C09132=1213.052,331.512,-71.588,-176.205,7.411,148.299
C09133=1213.056,331.264,-71.557,-176.207,7.408,148.299
C09134=1213.060,331.016,-71.525,-176.210,7.405,148.299
C09135=1213.064,330.768,-71.494,-176.212,7.402,148.299
C09136=1213.068,330.520,-71.463,-176.214,7.400,148.299
C09137=1213.073,330.272,-71.431,-176.216,7.396,148.298
C09138=1213.077,330.024,-71.400,-176.218,7.394,148.299
C09139=1213.081,329.776,-71.369,-176.220,7.391,148.298
C09140=1213.085,329.528,-71.338,-176.223,7.389,148.298
C09141=1213.089,329.280,-71.306,-176.225,7.385,148.298
C09142=1213.093,329.032,-71.275,-176.227,7.383,148.298
C09143=1213.098,328.784,-71.243,-176.229,7.380,148.298
C09144=1213.102,328.536,-71.212,-176.231,7.378,148.298
C09145=1213.106,328.288,-71.182,-176.233,7.374,148.298
C09146=1213.111,328.040,-71.150,-176.235,7.372,148.298
C09147=1213.115,327.792,-71.119,-176.238,7.369,148.298
C09148=1213.119,327.544,-71.087,-176.240,7.366,148.298
C09149=1213.123,327.296,-71.056,-176.242,7.363,148.297
C09150=1213.128,327.048,-71.026,-176.245,7.360,148.297
C09151=1213.132,326.800,-70.994,-176.246,7.358,148.297
C09152=1213.136,326.552,-70.963,-176.249,7.354,148.297
C09153=1213.141,326.304,-70.932,-176.251,7.352,148.297
C09154=1213.144,326.056,-70.900,-176.253,7.349,148.297
C09155=1213.148,325.808,-70.870,-176.255,7.347,148.297
C09156=1213.153,325.560,-70.839,-176.258,7.343,148.297
C09157=1213.157,325.311,-70.808,-176.260,7.341,148.297
C09158=1213.161,325.064,-70.777,-176.262,7.338,148.297
C09159=1213.165,324.815,-70.746,-176.264,7.336,148.297
C09160=1213.170,324.568,-70.715,-176.267,7.333,148.297
C09161=1213.174,324.320,-70.684,-176.268,7.330,148.297
C09162=1213.178,324.071,-70.653,-176.271,7.327,148.297
C09163=1213.182,323.824,-70.622,-176.273,7.325,148.297
C09164=1213.186,323.576,-70.591,-176.275,7.321,148.296
C09165=1213.191,323.327,-70.560,-176.277,7.319,148.296
C09166=1213.195,323.079,-70.530,-176.280,7.316,148.296
C09167=1213.199,322.831,-70.498,-176.282,7.313,148.296
C09168=1213.203,322.583,-70.468,-176.284,7.311,148.296
C09169=1213.207,322.336,-70.437,-176.287,7.307,148.296
C09170=1213.211,322.087,-70.406,-176.289,7.305,148.296
C09171=1213.216,321.839,-70.375,-176.291,7.302,148.296
C09172=1213.221,321.591,-70.344,-176.293,7.299,148.296
C09173=1213.224,321.343,-70.314,-176.296,7.296,148.296
C09174=1213.228,321.095,-70.283,-176.298,7.294,148.296
C09175=1213.233,320.847,-70.252,-176.300,7.291,148.296
C09176=1213.238,320.599,-70.221,-176.302,7.289,148.296
C09177=1213.241,320.351,-70.191,-176.305,7.286,148.296
C09178=1213.246,320.103,-70.160,-176.307,7.283,148.296
C09179=1213.250,319.855,-70.129,-176.309,7.280,148.296
C09180=1213.254,319.606,-70.098,-176.311,7.278,148.296
C09181=1213.258,319.358,-70.068,-176.314,7.275,148.296
C09182=1213.263,319.110,-70.037,-176.316,7.272,148.296
C09183=1213.267,318.862,-70.006,-176.318,7.269,148.296
C09184=1213.271,318.614,-69.976,-176.320,7.267,148.296
C09185=1213.275,318.366,-69.945,-176.323,7.264,148.296
C09186=1213.280,318.118,-69.914,-176.325,7.262,148.295
C09187=1213.284,317.870,-69.884,-176.327,7.258,148.295
C09188=1213.288,317.622,-69.853,-176.330,7.255,148.295
C09189=1213.293,317.373,-69.823,-176.332,7.253,148.295
C09190=1213.296,317.126,-69.793,-176.334,7.250,148.295
C09191=1213.301,316.878,-69.762,-176.336,7.248,148.295
C09192=1213.305,316.629,-69.731,-176.339,7.245,148.295
C09193=1213.309,316.381,-69.701,-176.341,7.242,148.295
C09194=1213.314,316.133,-69.670,-176.343,7.239,148.295
C09195=1213.318,315.885,-69.641,-176.346,7.237,148.295
C09196=1213.322,315.637,-69.610,-176.348,7.234,148.295
C09197=1213.327,315.361,-69.575,-176.351,7.231,148.295
C09198=1213.332,315.084,-69.542,-176.354,7.228,148.295
C09199=1213.336,314.809,-69.508,-176.356,7.226,148.295
C09200=1213.341,314.532,-69.474,-176.358,7.222,148.295
C09201=1213.345,314.284,-69.444,-176.361,7.219,148.295
C09202=1213.349,314.037,-69.413,-176.363,7.217,148.295
C09203=1213.354,313.789,-69.383,-176.365,7.214,148.295
C09204=1213.358,313.541,-69.353,-176.368,7.212,148.295
C09205=1213.363,313.293,-69.322,-176.370,7.209,148.295
C09206=1213.366,313.044,-69.292,-176.372,7.206,148.295
C09207=1213.371,312.796,-69.262,-176.375,7.203,148.295
C09208=1213.375,312.548,-69.232,-176.377,7.201,148.295
C09209=1213.379,312.300,-69.201,-176.379,7.198,148.295
C09210=1213.384,312.052,-69.171,-176.381,7.196,148.295
C09211=1213.388,311.804,-69.141,-176.384,7.193,148.295
C09212=1213.392,311.556,-69.111,-176.386,7.190,148.295
C09213=1213.396,311.307,-69.080,-176.389,7.187,148.295
C09214=1213.400,311.059,-69.050,-176.392,7.184,148.295
C09215=1213.405,310.811,-69.020,-176.393,7.182,148.295
C09216=1213.409,310.563,-68.990,-176.396,7.179,148.295
C09217=1213.413,310.315,-68.960,-176.398,7.177,148.295
C09218=1213.418,310.067,-68.929,-176.401,7.173,148.295
C09219=1213.422,309.819,-68.900,-176.403,7.171,148.295
C09220=1213.427,309.571,-68.869,-176.405,7.168,148.295
C09221=1213.431,309.322,-68.840,-176.408,7.166,148.295
C09222=1213.435,309.074,-68.809,-176.410,7.163,148.295
C09223=1213.440,308.826,-68.780,-176.412,7.161,148.295
C09224=1213.443,308.578,-68.749,-176.415,7.158,148.295
C09225=1213.448,308.329,-68.719,-176.417,7.156,148.295
C09226=1213.452,308.081,-68.689,-176.419,7.152,148.295
C09227=1213.456,307.833,-68.659,-176.421,7.150,148.295
C09228=1213.461,307.585,-68.629,-176.424,7.147,148.295
C09229=1213.465,307.337,-68.599,-176.426,7.145,148.295
C09230=1213.469,307.089,-68.570,-176.429,7.142,148.295
C09231=1213.473,306.841,-68.539,-176.431,7.140,148.295
C09232=1213.478,306.593,-68.509,-176.433,7.137,148.295
C09233=1213.482,306.344,-68.480,-176.436,7.134,148.295
C09234=1213.486,306.096,-68.449,-176.438,7.132,148.295
C09235=1213.491,305.848,-68.420,-176.441,7.129,148.295
C09236=1213.495,305.600,-68.390,-176.443,7.127,148.295
C09237=1213.499,305.352,-68.360,-176.445,7.124,148.295
C09238=1213.504,305.104,-68.330,-176.448,7.122,148.296
C09239=1213.508,304.855,-68.301,-176.450,7.119,148.296
C09240=1213.512,304.607,-68.271,-176.452,7.116,148.296
C09241=1213.517,304.359,-68.240,-176.455,7.113,148.296
C09242=1213.521,304.111,-68.211,-176.457,7.111,148.296
C09243=1213.525,303.862,-68.182,-176.460,7.108,148.296
C09244=1213.529,303.614,-68.152,-176.462,7.106,148.296
C09245=1213.534,303.366,-68.121,-176.465,7.103,148.296
C09246=1213.538,303.118,-68.092,-176.467,7.101,148.296
C09247=1213.542,302.870,-68.062,-176.469,7.098,148.296
C09248=1213.546,302.621,-68.033,-176.472,7.095,148.296
C09249=1213.550,302.373,-68.004,-176.474,7.092,148.296
C09250=1213.555,302.125,-67.973,-176.476,7.090,148.296
C09251=1213.559,301.877,-67.943,-176.479,7.087,148.296
C09252=1213.563,301.629,-67.914,-176.481,7.085,148.296
C09253=1213.568,301.380,-67.884,-176.484,7.082,148.296
C09254=1213.572,301.132,-67.855,-176.486,7.080,148.296
C09255=1213.577,300.885,-67.826,-176.489,7.077,148.296
C09256=1213.581,300.636,-67.796,-176.491,7.074,148.296
C09257=1213.586,300.388,-67.766,-176.494,7.072,148.296
C09258=1213.590,300.139,-67.737,-176.496,7.069,148.296
C09259=1213.594,299.891,-67.707,-176.498,7.067,148.297
C09260=1213.598,299.643,-67.678,-176.501,7.064,148.297
C09261=1213.602,299.395,-67.649,-176.503,7.062,148.297
C09262=1213.607,299.146,-67.619,-176.506,7.059,148.297
C09263=1213.611,298.898,-67.590,-176.508,7.057,148.297
C09264=1213.615,298.650,-67.560,-176.510,7.054,148.297
C09265=1213.619,298.402,-67.531,-176.513,7.052,148.297
C09266=1213.624,298.154,-67.502,-176.515,7.049,148.297
C09267=1213.628,297.906,-67.472,-176.517,7.046,148.297
C09268=1213.632,297.658,-67.443,-176.520,7.043,148.297
C09269=1213.636,297.409,-67.413,-176.523,7.041,148.297
C09270=1213.641,297.161,-67.383,-176.525,7.038,148.297
C09271=1213.646,296.912,-67.354,-176.527,7.036,148.297
C09272=1213.650,296.664,-67.324,-176.530,7.034,148.297
C09273=1213.655,296.416,-67.296,-176.532,7.031,148.297
C09274=1213.659,296.168,-67.267,-176.534,7.029,148.297
C09275=1213.662,295.920,-67.238,-176.537,7.026,148.297
C09276=1213.667,295.671,-67.208,-176.539,7.023,148.297
C09277=1213.671,295.423,-67.179,-176.542,7.021,148.298
C09278=1213.675,295.175,-67.149,-176.544,7.019,148.298
C09279=1213.679,294.926,-67.121,-176.547,7.016,148.298
C09280=1213.684,294.678,-67.091,-176.549,7.013,148.298
C09281=1213.688,294.430,-67.062,-176.551,7.011,148.298
C09282=1213.693,294.182,-67.033,-176.554,7.008,148.298
C09283=1213.697,293.934,-67.003,-176.557,7.006,148.298
C09284=1213.701,293.685,-66.974,-176.559,7.003,148.298
C09285=1213.706,293.437,-66.945,-176.561,7.001,148.298
C09286=1213.710,293.189,-66.916,-176.564,6.998,148.298
C09287=1213.715,292.940,-66.887,-176.566,6.996,148.298
C09288=1213.719,292.692,-66.858,-176.568,6.994,148.298
C09289=1213.723,292.445,-66.829,-176.572,6.991,148.299
C09290=1213.727,292.196,-66.800,-176.574,6.989,148.299
C09291=1213.732,291.947,-66.771,-176.576,6.986,148.299
C09292=1213.736,291.699,-66.741,-176.578,6.983,148.299
C09293=1213.740,291.450,-66.713,-176.581,6.980,148.299
C09294=1213.745,291.203,-66.684,-176.583,6.978,148.299
C09295=1213.748,290.955,-66.655,-176.586,6.976,148.299
C09296=1213.753,290.706,-66.626,-176.589,6.973,148.299
C09297=1213.757,290.458,-66.597,-176.591,6.971,148.299
C09298=1213.762,290.209,-66.568,-176.593,6.968,148.299
C09299=1213.766,289.961,-66.539,-176.596,6.966,148.300
C09300=1213.771,289.713,-66.509,-176.599,6.963,148.300
C09301=1213.775,289.438,-66.478,-176.601,6.961,148.300
C09302=1213.780,289.164,-66.446,-176.603,6.958,148.300
C09303=1213.785,288.890,-66.414,-176.607,6.955,148.300
C09304=1213.790,288.616,-66.382,-176.609,6.952,148.300
C09305=1213.795,288.368,-66.354,-176.611,6.950,148.300
C09306=1213.798,288.120,-66.325,-176.614,6.948,148.300
C09307=1213.803,287.871,-66.296,-176.617,6.945,148.300
C09308=1213.808,287.623,-66.268,-176.619,6.943,148.300
C09309=1213.812,287.375,-66.238,-176.621,6.940,148.300
C09310=1213.816,287.126,-66.210,-176.624,6.938,148.301
C09311=1213.820,286.878,-66.181,-176.626,6.936,148.301
C09312=1213.825,286.629,-66.152,-176.629,6.933,148.301
C09313=1213.828,286.382,-66.123,-176.631,6.930,148.301
C09314=1213.833,286.133,-66.095,-176.634,6.928,148.301
C09315=1213.838,285.884,-66.066,-176.636,6.925,148.301
C09316=1213.841,285.637,-66.037,-176.638,6.923,148.301
C09317=1213.846,285.388,-66.009,-176.642,6.921,148.301
C09318=1213.851,285.139,-65.980,-176.644,6.918,148.301
C09319=1213.854,284.891,-65.952,-176.646,6.915,148.301
C09320=1213.859,284.643,-65.923,-176.648,6.913,148.302
C09321=1213.864,284.394,-65.894,-176.651,6.911,148.302
C09322=1213.867,284.146,-65.866,-176.654,6.908,148.302
C09323=1213.872,283.898,-65.837,-176.656,6.906,148.302
C09324=1213.876,283.650,-65.809,-176.659,6.903,148.302
C09325=1213.881,283.402,-65.781,-176.661,6.901,148.302
C09326=1213.885,283.153,-65.751,-176.663,6.899,148.302
C09327=1213.889,282.905,-65.723,-176.666,6.896,148.302
C09328=1213.894,282.656,-65.695,-176.669,6.894,148.303
C09329=1213.898,282.408,-65.667,-176.671,6.892,148.303
C09330=1213.903,282.160,-65.638,-176.673,6.889,148.303
C09331=1213.907,281.912,-65.609,-176.676,6.887,148.303
C09332=1213.912,281.664,-65.581,-176.679,6.884,148.303
C09333=1213.916,281.415,-65.552,-176.681,6.882,148.303
C09334=1213.920,281.166,-65.524,-176.683,6.880,148.303
C09335=1213.925,280.918,-65.496,-176.686,6.877,148.303
C09336=1213.929,280.669,-65.468,-176.688,6.875,148.304
C09337=1213.934,280.421,-65.439,-176.691,6.873,148.304
C09338=1213.938,280.173,-65.411,-176.694,6.870,148.304
C09339=1213.942,279.925,-65.382,-176.696,6.867,148.304
C09340=1213.946,279.676,-65.354,-176.698,6.866,148.304
C09341=1213.950,279.429,-65.326,-176.701,6.863,148.304
C09342=1213.955,279.180,-65.297,-176.703,6.860,148.304
C09343=1213.959,278.932,-65.270,-176.706,6.858,148.305
C09344=1213.964,278.683,-65.241,-176.708,6.855,148.305
C09345=1213.968,278.435,-65.213,-176.710,6.853,148.305
C09346=1213.973,278.186,-65.184,-176.714,6.851,148.305
C09347=1213.977,277.938,-65.156,-176.716,6.848,148.305
C09348=1213.981,277.689,-65.128,-176.718,6.846,148.305
C09349=1213.986,277.442,-65.100,-176.721,6.843,148.305
C09350=1213.990,277.193,-65.072,-176.723,6.841,148.305
C09351=1213.995,276.945,-65.043,-176.726,6.839,148.306
C09352=1213.998,276.696,-65.015,-176.728,6.836,148.306
C09353=1214.003,276.448,-64.988,-176.731,6.834,148.306
C09354=1214.008,276.199,-64.960,-176.733,6.832,148.306
C09355=1214.012,275.951,-64.932,-176.736,6.829,148.306
C09356=1214.016,275.702,-64.903,-176.739,6.827,148.306
C09357=1214.021,275.454,-64.875,-176.741,6.825,148.306
C09358=1214.024,275.206,-64.847,-176.743,6.822,148.307
C09359=1214.030,274.957,-64.819,-176.746,6.820,148.307
C09360=1214.033,274.709,-64.791,-176.748,6.818,148.307
C09361=1214.038,274.460,-64.763,-176.751,6.815,148.307
C09362=1214.043,274.212,-64.735,-176.753,6.813,148.307
C09363=1214.047,273.964,-64.707,-176.755,6.811,148.307
C09364=1214.051,273.716,-64.679,-176.759,6.808,148.308
C09365=1214.055,273.467,-64.651,-176.761,6.806,148.308
C09366=1214.060,273.218,-64.623,-176.763,6.804,148.308
C09367=1214.064,272.970,-64.595,-176.766,6.801,148.308
C09368=1214.068,272.722,-64.567,-176.768,6.799,148.308
C09369=1214.073,272.474,-64.539,-176.771,6.797,148.308
C09370=1214.078,272.224,-64.512,-176.773,6.794,148.308
C09371=1214.082,271.977,-64.484,-176.776,6.792,148.309
C09372=1214.086,271.728,-64.456,-176.778,6.790,148.309
C09373=1214.090,271.480,-64.429,-176.781,6.788,148.309
C09374=1214.095,271.231,-64.400,-176.784,6.785,148.309
C09375=1214.099,270.983,-64.372,-176.786,6.783,148.309
C09376=1214.104,270.734,-64.345,-176.788,6.781,148.309
C09377=1214.108,270.486,-64.317,-176.791,6.778,148.309
C09378=1214.112,270.238,-64.289,-176.794,6.776,148.310
C09379=1214.117,269.989,-64.262,-176.796,6.774,148.310
C09380=1214.122,269.741,-64.234,-176.799,6.771,148.310
C09381=1214.126,269.492,-64.206,-176.801,6.769,148.310
C09382=1214.130,269.244,-64.179,-176.804,6.767,148.310
C09383=1214.134,268.996,-64.151,-176.806,6.765,148.311
C09384=1214.138,268.747,-64.123,-176.809,6.762,148.311
C09385=1214.144,268.499,-64.095,-176.811,6.760,148.311
C09386=1214.148,268.250,-64.068,-176.814,6.758,148.311
C09387=1214.152,268.002,-64.040,-176.816,6.755,148.311
C09388=1214.157,267.753,-64.013,-176.818,6.753,148.311
C09389=1214.161,267.505,-63.985,-176.821,6.751,148.312
C09390=1214.165,267.256,-63.958,-176.823,6.749,148.312
C09391=1214.169,267.008,-63.930,-176.826,6.746,148.312
C09392=1214.174,266.760,-63.903,-176.828,6.744,148.312
C09393=1214.178,266.511,-63.875,-176.831,6.742,148.312
C09394=1214.183,266.262,-63.847,-176.834,6.739,148.312
C09395=1214.188,266.015,-63.819,-176.836,6.737,148.313
C09396=1214.192,265.766,-63.792,-176.839,6.735,148.313
C09397=1214.196,265.517,-63.765,-176.841,6.733,148.313
C09398=1214.201,265.269,-63.737,-176.844,6.730,148.313
C09399=1214.205,265.020,-63.710,-176.846,6.728,148.313
C09400=1214.210,264.772,-63.683,-176.849,6.726,148.313
C09401=1214.214,264.523,-63.655,-176.851,6.724,148.314
C09402=1214.218,264.275,-63.628,-176.854,6.721,148.314
C09403=1214.223,264.027,-63.600,-176.856,6.719,148.314
C09404=1214.227,263.779,-63.573,-176.859,6.717,148.314
C09405=1214.231,263.505,-63.543,-176.862,6.714,148.314
C09406=1214.236,263.233,-63.512,-176.864,6.712,148.315
C09407=1214.241,262.960,-63.483,-176.867,6.709,148.315
C09408=1214.247,262.687,-63.453,-176.870,6.708,148.315
C09409=1214.251,262.439,-63.425,-176.873,6.705,148.315
C09410=1214.255,262.190,-63.398,-176.875,6.703,148.315
C09411=1214.260,261.942,-63.371,-176.878,6.701,148.316
C09412=1214.264,261.693,-63.344,-176.880,6.699,148.316
C09413=1214.269,261.445,-63.317,-176.883,6.696,148.316
C09414=1214.273,261.197,-63.289,-176.885,6.694,148.316
C09415=1214.277,260.948,-63.262,-176.888,6.692,148.316
C09416=1214.281,260.700,-63.235,-176.890,6.690,148.316
C09417=1214.286,260.451,-63.208,-176.893,6.687,148.317
C09418=1214.291,260.203,-63.181,-176.895,6.685,148.317
C09419=1214.295,259.955,-63.153,-176.898,6.683,148.317
C09420=1214.300,259.706,-63.126,-176.900,6.681,148.317
C09421=1214.304,259.457,-63.099,-176.903,6.678,148.317
C09422=1214.308,259.209,-63.072,-176.906,6.676,148.318
C09423=1214.312,258.960,-63.045,-176.908,6.674,148.318
C09424=1214.317,258.712,-63.018,-176.910,6.672,148.318
C09425=1214.322,258.463,-62.991,-176.913,6.670,148.318
C09426=1214.326,258.215,-62.964,-176.916,6.667,148.319
C09427=1214.331,257.966,-62.937,-176.918,6.665,148.319
C09428=1214.334,257.717,-62.910,-176.920,6.663,148.319
C09429=1214.339,257.469,-62.883,-176.923,6.661,148.319
C09430=1214.344,257.220,-62.856,-176.925,6.659,148.319
C09431=1214.348,256.972,-62.829,-176.928,6.656,148.320
C09432=1214.353,256.723,-62.802,-176.931,6.654,148.320
C09433=1214.357,256.475,-62.775,-176.933,6.652,148.320
C09434=1214.361,256.227,-62.748,-176.935,6.650,148.320
C09435=1214.366,255.978,-62.721,-176.938,6.647,148.320
C09436=1214.371,255.730,-62.694,-176.941,6.646,148.321
C09437=1214.375,255.482,-62.668,-176.943,6.643,148.321
C09438=1214.379,255.232,-62.640,-176.946,6.641,148.321
C09439=1214.383,254.984,-62.613,-176.948,6.639,148.321
C09440=1214.387,254.736,-62.587,-176.951,6.637,148.321
C09441=1214.392,254.487,-62.560,-176.954,6.635,148.322
C09442=1214.397,254.239,-62.532,-176.956,6.633,148.322
C09443=1214.401,253.990,-62.505,-176.958,6.631,148.322
C09444=1214.405,253.741,-62.480,-176.961,6.628,148.322
C09445=1214.410,253.493,-62.453,-176.963,6.627,148.322
C09446=1214.415,253.244,-62.426,-176.966,6.624,148.323
C09447=1214.419,252.996,-62.399,-176.969,6.622,148.323
C09448=1214.423,252.748,-62.372,-176.971,6.620,148.323
C09449=1214.428,252.499,-62.345,-176.973,6.618,148.323
C09450=1214.432,252.250,-62.319,-176.976,6.616,148.324
C09451=1214.437,252.002,-62.292,-176.979,6.613,148.324
C09452=1214.441,251.754,-62.266,-176.981,6.611,148.324
C09453=1214.445,251.505,-62.239,-176.984,6.609,148.324
C09454=1214.450,251.256,-62.212,-176.986,6.607,148.324
C09455=1214.454,251.008,-62.186,-176.989,6.605,148.325
C09456=1214.459,250.759,-62.159,-176.991,6.603,148.325
C09457=1214.463,250.511,-62.132,-176.994,6.600,148.325
C09458=1214.468,250.262,-62.106,-176.997,6.598,148.325
C09459=1214.473,250.014,-62.079,-176.999,6.596,148.326
C09460=1214.476,249.765,-62.052,-177.001,6.594,148.326
C09461=1214.481,249.516,-62.026,-177.004,6.592,148.326
C09462=1214.485,249.268,-62.000,-177.007,6.590,148.326
C09463=1214.490,249.020,-61.973,-177.009,6.587,148.326
C09464=1214.494,248.771,-61.947,-177.012,6.586,148.327
C09465=1214.499,248.522,-61.920,-177.014,6.584,148.327
C09466=1214.503,248.274,-61.894,-177.017,6.582,148.327
C09467=1214.508,248.025,-61.867,-177.019,6.580,148.327
C09468=1214.512,247.777,-61.840,-177.022,6.578,148.328
C09469=1214.517,247.528,-61.814,-177.024,6.576,148.328
C09470=1214.521,247.280,-61.788,-177.027,6.573,148.328
C09471=1214.526,247.030,-61.761,-177.030,6.571,148.328
C09472=1214.529,246.782,-61.735,-177.032,6.569,148.328
C09473=1214.535,246.534,-61.709,-177.035,6.567,148.329
C09474=1214.539,246.286,-61.682,-177.037,6.565,148.329
C09475=1214.544,246.037,-61.656,-177.039,6.563,148.329
C09476=1214.548,245.788,-61.630,-177.042,6.561,148.329
C09477=1214.553,245.539,-61.603,-177.045,6.558,148.330
C09478=1214.557,245.291,-61.577,-177.047,6.556,148.330
C09479=1214.561,245.042,-61.551,-177.050,6.554,148.330
C09480=1214.566,244.794,-61.524,-177.053,6.552,148.330
C09481=1214.570,244.545,-61.498,-177.055,6.550,148.331
C09482=1214.574,244.296,-61.471,-177.057,6.548,148.331
C09483=1214.579,244.048,-61.446,-177.060,6.547,148.331
C09484=1214.583,243.800,-61.420,-177.063,6.544,148.331
C09485=1214.588,243.551,-61.393,-177.065,6.542,148.332
C09486=1214.592,243.302,-61.367,-177.068,6.540,148.332
C09487=1214.597,243.054,-61.340,-177.070,6.538,148.332
C09488=1214.601,242.805,-61.314,-177.073,6.536,148.332
C09489=1214.605,242.556,-61.289,-177.075,6.534,148.333
C09490=1214.611,242.308,-61.262,-177.078,6.532,148.333
C09491=1214.615,242.060,-61.236,-177.080,6.530,148.333
C09492=1214.619,241.811,-61.210,-177.083,6.528,148.333
C09493=1214.624,241.562,-61.183,-177.086,6.525,148.334
C09494=1214.628,241.313,-61.158,-177.088,6.523,148.334
C09495=1214.632,241.065,-61.132,-177.091,6.521,148.334
C09496=1214.637,240.817,-61.106,-177.093,6.519,148.334
C09497=1214.642,240.568,-61.079,-177.096,6.518,148.335
C09498=1214.646,240.319,-61.054,-177.098,6.515,148.335
C09499=1214.650,240.070,-61.028,-177.101,6.514,148.335
C09500=1214.655,239.821,-61.002,-177.103,6.512,148.335
C09501=1214.660,239.574,-60.975,-177.105,6.509,148.335
C09502=1214.664,239.325,-60.950,-177.109,6.507,148.336
C09503=1214.668,239.076,-60.924,-177.111,6.505,148.336
C09504=1214.673,238.827,-60.898,-177.114,6.503,148.336
C09505=1214.677,238.578,-60.872,-177.116,6.501,148.336
C09506=1214.682,238.330,-60.846,-177.119,6.499,148.337
C09507=1214.686,238.082,-60.820,-177.121,6.497,148.337
C09508=1214.690,237.833,-60.794,-177.124,6.495,148.337
C09509=1214.696,237.562,-60.766,-177.126,6.493,148.337
C09510=1214.701,237.290,-60.738,-177.129,6.490,148.338
C09511=1214.705,237.019,-60.709,-177.132,6.489,148.338
C09512=1214.711,236.747,-60.682,-177.135,6.486,148.338
C09513=1214.715,236.499,-60.656,-177.138,6.484,148.339
C09514=1214.719,236.250,-60.630,-177.140,6.482,148.339
C09515=1214.724,236.002,-60.605,-177.142,6.480,148.339
C09516=1214.728,235.753,-60.579,-177.145,6.478,148.339
C09517=1214.733,235.504,-60.553,-177.148,6.476,148.340
C09518=1214.737,235.255,-60.527,-177.150,6.474,148.340
C09519=1214.742,235.007,-60.501,-177.152,6.472,148.340
C09520=1214.746,234.758,-60.476,-177.155,6.470,148.340
C09521=1214.751,234.509,-60.450,-177.158,6.469,148.341
C09522=1214.755,234.261,-60.425,-177.160,6.467,148.341
C09523=1214.760,234.012,-60.399,-177.163,6.465,148.341
C09524=1214.764,233.763,-60.373,-177.165,6.463,148.342
C09525=1214.769,233.515,-60.348,-177.168,6.460,148.342
C09526=1214.773,233.267,-60.322,-177.171,6.458,148.342
C09527=1214.778,233.017,-60.296,-177.173,6.456,148.342
C09528=1214.783,232.769,-60.270,-177.176,6.454,148.343
C09529=1214.787,232.521,-60.244,-177.178,6.452,148.343
C09530=1214.791,232.272,-60.219,-177.181,6.450,148.343
C09531=1214.796,232.024,-60.193,-177.183,6.448,148.344
C09532=1214.800,231.775,-60.167,-177.186,6.447,148.344
C09533=1214.805,231.525,-60.142,-177.188,6.444,148.344
C09534=1214.810,231.277,-60.117,-177.191,6.443,148.344
C09535=1214.814,231.029,-60.091,-177.193,6.441,148.345
C09536=1214.818,230.780,-60.066,-177.196,6.439,148.345
C09537=1214.823,230.532,-60.040,-177.199,6.437,148.345
C09538=1214.827,230.282,-60.015,-177.201,6.435,148.345
C09539=1214.832,230.033,-59.989,-177.204,6.433,148.346
C09540=1214.837,229.785,-59.964,-177.206,6.431,148.346
C09541=1214.841,229.536,-59.938,-177.209,6.429,148.346
C09542=1214.846,229.288,-59.913,-177.211,6.427,148.347
C09543=1214.850,229.039,-59.888,-177.214,6.425,148.347
C09544=1214.854,228.790,-59.863,-177.216,6.423,148.347
C09545=1214.858,228.542,-59.837,-177.219,6.421,148.347
C09546=1214.863,228.293,-59.812,-177.222,6.419,148.348
C09547=1214.868,228.045,-59.787,-177.225,6.417,148.348
C09548=1214.872,227.796,-59.761,-177.227,6.415,148.348
C09549=1214.877,227.547,-59.736,-177.229,6.413,148.348
C09550=1214.881,227.298,-59.711,-177.232,6.411,148.349
C09551=1214.886,227.050,-59.685,-177.235,6.409,148.349
C09552=1214.891,226.801,-59.660,-177.237,6.407,148.349
C09553=1214.895,226.552,-59.635,-177.240,6.406,148.350
C09554=1214.899,226.304,-59.610,-177.243,6.404,148.350
C09555=1214.904,226.055,-59.585,-177.245,6.402,148.350
C09556=1214.908,225.807,-59.559,-177.247,6.400,148.350
C09557=1214.913,225.557,-59.534,-177.250,6.398,148.351
C09558=1214.918,225.309,-59.509,-177.253,6.396,148.351
C09559=1214.922,225.060,-59.483,-177.255,6.394,148.351
C09560=1214.926,224.812,-59.459,-177.258,6.392,148.352
C09561=1214.931,224.563,-59.433,-177.260,6.390,148.352
C09562=1214.936,224.315,-59.409,-177.263,6.388,148.352
C09563=1214.940,224.066,-59.383,-177.265,6.386,148.353
C09564=1214.945,223.817,-59.358,-177.268,6.385,148.353
C09565=1214.949,223.569,-59.333,-177.271,6.383,148.353
C09566=1214.954,223.320,-59.308,-177.273,6.381,148.354
C09567=1214.958,223.071,-59.283,-177.276,6.379,148.354
C09568=1214.963,222.822,-59.258,-177.278,6.377,148.354
C09569=1214.967,222.573,-59.232,-177.281,6.375,148.354
C09570=1214.972,222.325,-59.208,-177.283,6.373,148.355
C09571=1214.976,222.076,-59.183,-177.286,6.371,148.355
C09572=1214.981,221.828,-59.158,-177.288,6.369,148.355
C09573=1214.985,221.578,-59.133,-177.291,6.368,148.356
C09574=1214.990,221.330,-59.108,-177.294,6.366,148.356
C09575=1214.994,221.081,-59.083,-177.296,6.364,148.356
C09576=1214.999,220.832,-59.058,-177.299,6.362,148.356
C09577=1215.003,220.584,-59.033,-177.301,6.360,148.357
C09578=1215.008,220.335,-59.008,-177.304,6.358,148.357
C09579=1215.012,220.086,-58.983,-177.306,6.356,148.357
C09580=1215.017,219.838,-58.959,-177.309,6.354,148.358
C09581=1215.022,219.589,-58.934,-177.312,6.352,148.358
C09582=1215.026,219.340,-58.909,-177.314,6.351,148.358
C09583=1215.030,219.092,-58.884,-177.317,6.349,148.359
C09584=1215.035,218.842,-58.859,-177.320,6.347,148.359
C09585=1215.039,218.594,-58.835,-177.322,6.345,148.359
C09586=1215.044,218.346,-58.810,-177.324,6.343,148.359
C09587=1215.049,218.096,-58.785,-177.327,6.341,148.360
C09588=1215.053,217.848,-58.760,-177.330,6.339,148.360
C09589=1215.057,217.599,-58.735,-177.332,6.337,148.360
C09590=1215.062,217.350,-58.710,-177.335,6.336,148.361
C09591=1215.067,217.102,-58.686,-177.338,6.334,148.361
C09592=1215.071,216.853,-58.661,-177.340,6.332,148.361
C09593=1215.076,216.604,-58.637,-177.343,6.330,148.362
C09594=1215.080,216.355,-58.612,-177.345,6.328,148.362
C09595=1215.085,216.106,-58.588,-177.348,6.326,148.362
C09596=1215.089,215.858,-58.562,-177.350,6.324,148.363
C09597=1215.093,215.609,-58.538,-177.353,6.322,148.363
C09598=1215.098,215.360,-58.513,-177.356,6.320,148.363
C09599=1215.103,215.112,-58.489,-177.358,6.319,148.364
C09600=1215.107,214.863,-58.464,-177.361,6.317,148.364
C09601=1215.112,214.614,-58.439,-177.363,6.315,148.364
C09602=1215.117,214.365,-58.415,-177.366,6.313,148.365
C09603=1215.121,214.116,-58.390,-177.369,6.311,148.365
C09604=1215.126,213.868,-58.366,-177.371,6.309,148.365
C09605=1215.130,213.620,-58.341,-177.374,6.308,148.366
C09606=1215.134,213.370,-58.316,-177.377,6.306,148.366
C09607=1215.139,213.122,-58.292,-177.379,6.304,148.366
C09608=1215.144,212.873,-58.268,-177.382,6.302,148.367
C09609=1215.148,212.624,-58.243,-177.385,6.300,148.367
C09610=1215.153,212.375,-58.219,-177.387,6.298,148.367
C09611=1215.157,212.127,-58.195,-177.390,6.296,148.368
C09612=1215.162,211.878,-58.170,-177.392,6.295,148.368
C09613=1215.167,211.607,-58.144,-177.395,6.293,148.368
C09614=1215.172,211.337,-58.117,-177.398,6.291,148.369
C09615=1215.177,211.067,-58.091,-177.400,6.289,148.369
C09616=1215.182,210.797,-58.064,-177.403,6.287,148.369
C09617=1215.186,210.548,-58.040,-177.406,6.285,148.370
C09618=1215.191,210.298,-58.016,-177.408,6.284,148.370
C09619=1215.195,210.050,-57.992,-177.411,6.282,148.370
C09620=1215.201,209.801,-57.967,-177.414,6.280,148.371
C09621=1215.204,209.552,-57.942,-177.416,6.278,148.371
C09622=1215.209,209.304,-57.918,-177.419,6.276,148.371
C09623=1215.214,209.055,-57.894,-177.422,6.274,148.372
C09624=1215.218,208.806,-57.870,-177.424,6.272,148.372
C09625=1215.223,208.558,-57.846,-177.427,6.271,148.372
C09626=1215.228,208.308,-57.821,-177.429,6.269,148.373
C09627=1215.232,208.060,-57.797,-177.432,6.267,148.373
C09628=1215.236,207.811,-57.773,-177.435,6.265,148.373
C09629=1215.241,207.562,-57.748,-177.437,6.263,148.374
C09630=1215.245,207.313,-57.724,-177.439,6.262,148.374
C09631=1215.250,207.064,-57.701,-177.442,6.260,148.374
C09632=1215.255,206.815,-57.676,-177.445,6.259,148.375
C09633=1215.259,206.567,-57.652,-177.447,6.257,148.375
C09634=1215.264,206.318,-57.628,-177.450,6.255,148.375
C09635=1215.269,206.070,-57.604,-177.452,6.253,148.375
C09636=1215.273,205.820,-57.579,-177.455,6.251,148.376
C09637=1215.277,205.572,-57.555,-177.457,6.249,148.376
C09638=1215.282,205.323,-57.532,-177.460,6.247,148.376
C09639=1215.287,205.074,-57.508,-177.463,6.245,148.377
C09640=1215.292,204.826,-57.483,-177.465,6.244,148.377
C09641=1215.296,204.577,-57.460,-177.468,6.242,148.377
C09642=1215.300,204.327,-57.435,-177.470,6.241,148.378
C09643=1215.305,204.079,-57.411,-177.473,6.239,148.378
C09644=1215.309,203.830,-57.388,-177.475,6.237,148.378
C09645=1215.314,203.581,-57.363,-177.478,6.235,148.379
C09646=1215.319,203.332,-57.340,-177.481,6.233,148.379
C09647=1215.324,203.084,-57.316,-177.483,6.232,148.379
C09648=1215.328,202.835,-57.292,-177.486,6.230,148.380
C09649=1215.332,202.586,-57.268,-177.489,6.228,148.380
C09650=1215.337,202.337,-57.243,-177.491,6.226,148.381
C09651=1215.342,202.088,-57.220,-177.494,6.224,148.381
C09652=1215.346,201.840,-57.196,-177.496,6.223,148.381
C09653=1215.351,201.591,-57.173,-177.499,6.222,148.382
C09654=1215.355,201.342,-57.149,-177.502,6.220,148.382
C09655=1215.360,201.093,-57.125,-177.504,6.218,148.382
C09656=1215.364,200.845,-57.101,-177.507,6.216,148.383
C09657=1215.369,200.596,-57.078,-177.510,6.214,148.383
C09658=1215.374,200.347,-57.053,-177.512,6.212,148.384
C09659=1215.378,200.097,-57.029,-177.515,6.211,148.384
C09660=1215.383,199.849,-57.005,-177.517,6.210,148.384
C09661=1215.387,199.600,-56.982,-177.520,6.208,148.385
C09662=1215.392,199.351,-56.958,-177.522,6.206,148.385
C09663=1215.397,199.102,-56.934,-177.525,6.204,148.385
C09664=1215.401,198.854,-56.910,-177.528,6.202,148.386
C09665=1215.406,198.605,-56.887,-177.530,6.200,148.386
C09666=1215.410,198.356,-56.864,-177.533,6.199,148.386
C09667=1215.415,198.107,-56.840,-177.536,6.197,148.387
C09668=1215.419,197.858,-56.816,-177.538,6.196,148.387
C09669=1215.424,197.609,-56.793,-177.540,6.194,148.387
C09670=1215.429,197.361,-56.769,-177.543,6.192,148.388
C09671=1215.433,197.112,-56.745,-177.546,6.190,148.388
C09672=1215.438,196.863,-56.722,-177.548,6.188,148.388
C09673=1215.442,196.614,-56.698,-177.551,6.187,148.389
C09674=1215.447,196.365,-56.675,-177.554,6.185,148.389
C09675=1215.452,196.116,-56.651,-177.556,6.184,148.389
C09676=1215.456,195.868,-56.627,-177.558,6.182,148.390
C09677=1215.461,195.619,-56.604,-177.561,6.180,148.390
C09678=1215.466,195.370,-56.580,-177.564,6.178,148.390
C09679=1215.470,195.121,-56.557,-177.567,6.177,148.391
C09680=1215.475,194.872,-56.533,-177.569,6.175,148.391
C09681=1215.479,194.623,-56.510,-177.572,6.173,148.392
C09682=1215.484,194.374,-56.486,-177.574,6.172,148.392
C09683=1215.489,194.125,-56.463,-177.577,6.170,148.392
C09684=1215.493,193.876,-56.440,-177.579,6.168,148.393
C09685=1215.498,193.628,-56.416,-177.582,6.167,148.393
C09686=1215.502,193.379,-56.393,-177.585,6.165,148.394
C09687=1215.506,193.130,-56.369,-177.587,6.163,148.394
C09688=1215.511,192.881,-56.346,-177.589,6.162,148.394
C09689=1215.516,192.632,-56.323,-177.592,6.160,148.395
C09690=1215.521,192.383,-56.299,-177.595,6.158,148.395
C09691=1215.525,192.135,-56.275,-177.597,6.156,148.395
C09692=1215.530,191.886,-56.252,-177.600,6.155,148.396
C09693=1215.535,191.637,-56.229,-177.603,6.154,148.396
C09694=1215.539,191.389,-56.206,-177.605,6.152,148.397
C09695=1215.544,191.140,-56.183,-177.608,6.150,148.397
C09696=1215.548,190.891,-56.159,-177.610,6.148,148.397
C09697=1215.553,190.641,-56.136,-177.613,6.147,148.398
C09698=1215.558,190.392,-56.113,-177.616,6.145,148.398
C09699=1215.562,190.143,-56.089,-177.618,6.144,148.398
C09700=1215.566,189.895,-56.067,-177.621,6.142,148.399
C09701=1215.571,189.646,-56.043,-177.623,6.140,148.399
C09702=1215.576,189.397,-56.020,-177.626,6.138,148.399
C09703=1215.581,189.148,-55.997,-177.628,6.136,148.400
C09704=1215.585,188.900,-55.974,-177.631,6.135,148.400
C09705=1215.590,188.651,-55.951,-177.634,6.134,148.401
C09706=1215.594,188.402,-55.927,-177.636,6.132,148.401
C09707=1215.599,188.152,-55.904,-177.639,6.130,148.401
C09708=1215.603,187.904,-55.881,-177.642,6.128,148.402
C09709=1215.608,187.655,-55.858,-177.644,6.127,148.402
C09710=1215.613,187.406,-55.835,-177.646,6.126,148.402
C09711=1215.618,187.157,-55.812,-177.649,6.124,148.403
C09712=1215.622,186.909,-55.789,-177.652,6.122,148.403
C09713=1215.626,186.660,-55.765,-177.654,6.120,148.404
C09714=1215.631,186.410,-55.743,-177.657,6.119,148.404
C09715=1215.635,186.161,-55.720,-177.660,6.118,148.404
C09716=1215.641,185.913,-55.697,-177.662,6.116,148.405
C09717=1215.646,185.643,-55.672,-177.665,6.114,148.405
C09718=1215.651,185.374,-55.648,-177.668,6.112,148.406
C09719=1215.656,185.104,-55.623,-177.671,6.111,148.406
C09720=1215.661,184.835,-55.597,-177.673,6.109,148.406
C09721=1215.665,184.585,-55.575,-177.676,6.107,148.407
C09722=1215.670,184.336,-55.551,-177.679,6.105,148.407
C09723=1215.675,184.087,-55.528,-177.681,6.104,148.408
C09724=1215.679,183.839,-55.505,-177.684,6.103,148.408
C09725=1215.684,183.590,-55.483,-177.687,6.101,148.408
C09726=1215.688,183.341,-55.460,-177.689,6.099,148.409
C09727=1215.693,183.092,-55.437,-177.691,6.098,148.409
C09728=1215.698,182.843,-55.414,-177.694,6.096,148.410
C09729=1215.702,182.594,-55.392,-177.697,6.094,148.410
C09730=1215.707,182.345,-55.368,-177.699,6.093,148.410
C09731=1215.711,182.097,-55.346,-177.701,6.092,148.411
C09732=1215.716,181.847,-55.323,-177.704,6.090,148.411
C09733=1215.721,181.599,-55.300,-177.707,6.088,148.412
C09734=1215.725,181.350,-55.277,-177.710,6.086,148.412
C09735=1215.730,181.100,-55.255,-177.712,6.085,148.412
C09736=1215.734,180.851,-55.232,-177.714,6.084,148.413
C09737=1215.740,180.603,-55.209,-177.717,6.082,148.413
C09738=1215.744,180.354,-55.187,-177.720,6.080,148.413
C09739=1215.749,180.105,-55.163,-177.722,6.079,148.414
C09740=1215.753,179.856,-55.141,-177.725,6.077,148.414
C09741=1215.758,179.607,-55.118,-177.728,6.076,148.415
C09742=1215.762,179.358,-55.096,-177.730,6.074,148.415
C09743=1215.767,179.109,-55.073,-177.732,6.073,148.415
C09744=1215.772,178.861,-55.051,-177.735,6.071,148.416
C09745=1215.777,178.611,-55.028,-177.738,6.070,148.416
C09746=1215.781,178.362,-55.005,-177.741,6.068,148.417
C09747=1215.786,178.114,-54.982,-177.743,6.067,148.417
C09748=1215.790,177.865,-54.960,-177.746,6.065,148.417
C09749=1215.795,177.616,-54.937,-177.748,6.063,148.418
C09750=1215.799,177.366,-54.915,-177.751,6.061,148.418
C09751=1215.804,177.118,-54.892,-177.754,6.061,148.419
C09752=1215.809,176.869,-54.870,-177.756,6.059,148.419
C09753=1215.813,176.620,-54.847,-177.759,6.057,148.420
C09754=1215.818,176.371,-54.825,-177.761,6.056,148.420
C09755=1215.823,176.122,-54.803,-177.764,6.054,148.420
C09756=1215.828,175.873,-54.780,-177.767,6.053,148.421
C09757=1215.832,175.624,-54.758,-177.769,6.051,148.421
C09758=1215.836,175.375,-54.735,-177.771,6.050,148.422
C09759=1215.842,175.126,-54.713,-177.774,6.048,148.422
C09760=1215.846,174.878,-54.690,-177.777,6.046,148.422
C09761=1215.850,174.628,-54.668,-177.779,6.045,148.423
C09762=1215.856,174.379,-54.645,-177.782,6.044,148.423
C09763=1215.860,174.130,-54.623,-177.785,6.042,148.424
C09764=1215.865,173.882,-54.600,-177.787,6.040,148.424
C09765=1215.869,173.632,-54.578,-177.789,6.039,148.424
C09766=1215.873,173.383,-54.556,-177.792,6.037,148.425
C09767=1215.879,173.135,-54.533,-177.795,6.036,148.425
C09768=1215.883,172.885,-54.511,-177.797,6.035,148.426
C09769=1215.888,172.637,-54.489,-177.800,6.033,148.426
C09770=1215.892,172.388,-54.467,-177.803,6.031,148.426
C09771=1215.897,172.138,-54.444,-177.805,6.030,148.427
C09772=1215.902,171.890,-54.423,-177.808,6.029,148.427
C09773=1215.906,171.641,-54.400,-177.811,6.027,148.428
C09774=1215.912,171.392,-54.377,-177.813,6.026,148.428
C09775=1215.916,171.143,-54.355,-177.815,6.024,148.429
C09776=1215.921,170.894,-54.334,-177.818,6.022,148.429
C09777=1215.925,170.645,-54.311,-177.821,6.021,148.429
C09778=1215.930,170.396,-54.289,-177.823,6.020,148.430
C09779=1215.935,170.147,-54.267,-177.826,6.018,148.430
C09780=1215.939,169.898,-54.245,-177.829,6.016,148.431
C09781=1215.944,169.649,-54.223,-177.831,6.015,148.431
C09782=1215.948,169.400,-54.200,-177.834,6.014,148.432
C09783=1215.953,169.151,-54.178,-177.836,6.012,148.432
C09784=1215.958,168.902,-54.156,-177.839,6.011,148.432
C09785=1215.962,168.653,-54.134,-177.841,6.009,148.433
C09786=1215.967,168.404,-54.112,-177.844,6.008,148.433
C09787=1215.972,168.155,-54.090,-177.846,6.007,148.434
C09788=1215.977,167.906,-54.068,-177.849,6.005,148.434
C09789=1215.981,167.658,-54.045,-177.852,6.003,148.434
C09790=1215.985,167.408,-54.023,-177.854,6.002,148.435
C09791=1215.990,167.160,-54.002,-177.857,6.000,148.435
C09792=1215.995,166.910,-53.979,-177.860,5.999,148.436
C09793=1216.000,166.661,-53.957,-177.862,5.998,148.436
C09794=1216.004,166.412,-53.935,-177.865,5.996,148.437
C09795=1216.009,166.163,-53.914,-177.868,5.994,148.437
C09796=1216.013,165.914,-53.892,-177.870,5.993,148.437
C09797=1216.018,165.665,-53.870,-177.872,5.992,148.438
C09798=1216.023,165.416,-53.848,-177.876,5.990,148.438
C09799=1216.027,165.167,-53.826,-177.878,5.989,148.439
C09800=1216.032,164.919,-53.804,-177.880,5.987,148.439
C09801=1216.037,164.669,-53.782,-177.882,5.986,148.440
C09802=1216.042,164.420,-53.760,-177.886,5.985,148.440
C09803=1216.047,164.171,-53.738,-177.888,5.983,148.440
C09804=1216.051,163.922,-53.716,-177.890,5.982,148.441
C09805=1216.056,163.673,-53.694,-177.893,5.980,148.441
C09806=1216.061,163.424,-53.673,-177.896,5.979,148.442
C09807=1216.065,163.175,-53.651,-177.898,5.978,148.442
C09808=1216.070,162.926,-53.629,-177.901,5.976,148.443
C09809=1216.075,162.677,-53.608,-177.904,5.974,148.443
C09810=1216.079,162.428,-53.586,-177.906,5.973,148.444
C09811=1216.084,162.179,-53.564,-177.909,5.972,148.444
C09812=1216.088,161.930,-53.542,-177.911,5.971,148.444
C09813=1216.093,161.681,-53.521,-177.914,5.969,148.445
C09814=1216.098,161.433,-53.499,-177.917,5.967,148.445
C09815=1216.102,161.183,-53.477,-177.919,5.966,148.446
C09816=1216.107,160.934,-53.456,-177.921,5.965,148.446
C09817=1216.112,160.685,-53.434,-177.924,5.963,148.446
C09818=1216.117,160.436,-53.412,-177.927,5.962,148.447
C09819=1216.121,160.187,-53.390,-177.929,5.960,148.447
C09820=1216.126,159.938,-53.368,-177.932,5.959,148.448
C09821=1216.131,159.669,-53.345,-177.935,5.958,148.448
C09822=1216.136,159.400,-53.322,-177.937,5.956,148.449
C09823=1216.141,159.131,-53.298,-177.940,5.955,148.449
C09824=1216.146,158.862,-53.275,-177.943,5.953,148.450
C09825=1216.151,158.613,-53.254,-177.945,5.952,148.450
C09826=1216.156,158.364,-53.233,-177.948,5.950,148.451
C09827=1216.160,158.115,-53.211,-177.951,5.949,148.451
C09828=1216.165,157.866,-53.189,-177.953,5.948,148.451
C09829=1216.170,157.617,-53.168,-177.956,5.946,148.452
C09830=1216.174,157.367,-53.146,-177.958,5.945,148.452
C09831=1216.179,157.119,-53.124,-177.961,5.943,148.453
C09832=1216.184,156.870,-53.103,-177.964,5.942,148.453
C09833=1216.188,156.620,-53.082,-177.966,5.941,148.454
C09834=1216.193,156.372,-53.060,-177.969,5.939,148.454
C09835=1216.198,156.123,-53.039,-177.971,5.938,148.455
C09836=1216.202,155.873,-53.017,-177.974,5.937,148.455
C09837=1216.207,155.625,-52.996,-177.977,5.935,148.456
C09838=1216.212,155.375,-52.975,-177.979,5.934,148.456
C09839=1216.217,155.127,-52.953,-177.982,5.932,148.457
C09840=1216.221,154.877,-52.932,-177.984,5.931,148.457
C09841=1216.226,154.628,-52.910,-177.987,5.930,148.457
C09842=1216.231,154.380,-52.889,-177.990,5.929,148.458
C09843=1216.236,154.130,-52.868,-177.992,5.927,148.458
C09844=1216.240,153.881,-52.846,-177.995,5.925,148.459
C09845=1216.245,153.632,-52.825,-177.997,5.925,148.459
C09846=1216.250,153.384,-52.804,-178.000,5.923,148.460
C09847=1216.255,153.134,-52.783,-178.002,5.922,148.460
C09848=1216.259,152.885,-52.761,-178.005,5.920,148.461
C09849=1216.263,152.636,-52.740,-178.008,5.919,148.461
C09850=1216.268,152.387,-52.719,-178.010,5.918,148.461
C09851=1216.274,152.138,-52.698,-178.013,5.916,148.462
C09852=1216.278,151.889,-52.676,-178.015,5.915,148.462
C09853=1216.282,151.640,-52.655,-178.018,5.913,148.463
C09854=1216.287,151.391,-52.634,-178.021,5.913,148.463
C09855=1216.292,151.142,-52.613,-178.023,5.911,148.464
C09856=1216.297,150.893,-52.592,-178.026,5.910,148.464
C09857=1216.301,150.644,-52.570,-178.029,5.908,148.465
C09858=1216.306,150.394,-52.549,-178.031,5.907,148.465
C09859=1216.311,150.146,-52.528,-178.033,5.906,148.466
C09860=1216.315,149.897,-52.507,-178.037,5.904,148.466
C09861=1216.321,149.647,-52.486,-178.039,5.903,148.467
C09862=1216.325,149.398,-52.464,-178.041,5.901,148.467
C09863=1216.329,149.149,-52.444,-178.044,5.901,148.468
C09864=1216.335,148.900,-52.423,-178.047,5.899,148.468
C09865=1216.339,148.651,-52.401,-178.049,5.898,148.468
C09866=1216.344,148.402,-52.381,-178.052,5.897,148.469
C09867=1216.348,148.152,-52.359,-178.054,5.896,148.469
C09868=1216.353,147.904,-52.338,-178.057,5.894,148.470
C09869=1216.358,147.655,-52.317,-178.059,5.893,148.470
C09870=1216.363,147.406,-52.296,-178.062,5.891,148.471
C09871=1216.368,147.156,-52.275,-178.065,5.890,148.471
C09872=1216.372,146.908,-52.254,-178.067,5.889,148.472
C09873=1216.377,146.659,-52.233,-178.070,5.887,148.472
C09874=1216.381,146.409,-52.213,-178.072,5.886,148.472
C09875=1216.386,146.160,-52.192,-178.075,5.885,148.473
C09876=1216.390,145.911,-52.171,-178.077,5.884,148.473
C09877=1216.396,145.662,-52.150,-178.080,5.882,148.474
C09878=1216.401,145.413,-52.129,-178.083,5.881,148.475
C09879=1216.405,145.164,-52.108,-178.085,5.879,148.475
C09880=1216.410,144.915,-52.087,-178.088,5.879,148.476
C09881=1216.415,144.666,-52.066,-178.090,5.877,148.476
C09882=1216.419,144.416,-52.045,-178.093,5.876,148.476
C09883=1216.424,144.167,-52.025,-178.096,5.875,148.477
C09884=1216.429,143.918,-52.004,-178.098,5.874,148.477
C09885=1216.433,143.669,-51.983,-178.101,5.872,148.478
C09886=1216.438,143.420,-51.962,-178.103,5.871,148.478
C09887=1216.443,143.172,-51.941,-178.106,5.869,148.479
C09888=1216.448,142.922,-51.920,-178.108,5.869,148.479
C09889=1216.452,142.673,-51.900,-178.111,5.867,148.480
C09890=1216.457,142.424,-51.879,-178.113,5.866,148.480
C09891=1216.462,142.175,-51.858,-178.116,5.865,148.481
C09892=1216.467,141.926,-51.837,-178.118,5.864,148.481
C09893=1216.471,141.677,-51.817,-178.122,5.862,148.482
C09894=1216.477,141.428,-51.796,-178.124,5.861,148.482
C09895=1216.481,141.179,-51.776,-178.126,5.859,148.482
C09896=1216.486,140.929,-51.754,-178.129,5.859,148.483
C09897=1216.490,140.680,-51.734,-178.132,5.857,148.483
C09898=1216.494,140.431,-51.714,-178.134,5.856,148.484
C09899=1216.500,140.182,-51.693,-178.137,5.854,148.484
C09900=1216.504,139.933,-51.672,-178.139,5.853,148.485
C09901=1216.509,139.684,-51.651,-178.142,5.852,148.485
C09902=1216.514,139.435,-51.631,-178.144,5.851,148.486
C09903=1216.519,139.185,-51.610,-178.148,5.850,148.487
C09904=1216.523,138.936,-51.590,-178.150,5.849,148.487
C09905=1216.528,138.687,-51.569,-178.152,5.847,148.487
C09906=1216.533,138.438,-51.548,-178.155,5.846,148.488
C09907=1216.537,138.189,-51.528,-178.158,5.844,148.488
C09908=1216.542,137.940,-51.508,-178.160,5.844,148.489
C09909=1216.547,137.691,-51.487,-178.163,5.842,148.489
C09910=1216.551,137.442,-51.466,-178.165,5.841,148.490
C09911=1216.556,137.192,-51.447,-178.168,5.840,148.490
C09912=1216.561,136.943,-51.426,-178.170,5.839,148.491
C09913=1216.566,136.694,-51.405,-178.173,5.837,148.491
C09914=1216.571,136.445,-51.384,-178.176,5.836,148.492
C09915=1216.575,136.196,-51.364,-178.179,5.835,148.492
C09916=1216.580,135.948,-51.344,-178.181,5.834,148.493
C09917=1216.585,135.699,-51.324,-178.183,5.832,148.493
C09918=1216.590,135.449,-51.303,-178.186,5.831,148.494
C09919=1216.595,135.200,-51.283,-178.188,5.830,148.494
C09920=1216.599,134.951,-51.263,-178.191,5.829,148.495
C09921=1216.604,134.702,-51.242,-178.193,5.828,148.495
C09922=1216.609,134.452,-51.222,-178.197,5.826,148.496
C09923=1216.613,134.203,-51.202,-178.199,5.826,148.496
C09924=1216.618,133.954,-51.181,-178.201,5.824,148.497
C09925=1216.623,133.686,-51.159,-178.204,5.823,148.497
C09926=1216.629,133.417,-51.137,-178.207,5.822,148.498
C09927=1216.634,133.149,-51.115,-178.210,5.820,148.498
C09928=1216.639,132.879,-51.093,-178.212,5.819,148.499
C09929=1216.643,132.630,-51.073,-178.215,5.817,148.499
C09930=1216.648,132.382,-51.054,-178.218,5.817,148.500
C09931=1216.654,132.132,-51.033,-178.220,5.815,148.500
C09932=1216.658,131.883,-51.012,-178.223,5.814,148.501
C09933=1216.663,131.634,-50.993,-178.225,5.813,148.501
C09934=1216.667,131.385,-50.972,-178.228,5.812,148.502
C09935=1216.672,131.136,-50.952,-178.230,5.811,148.502
C09936=1216.677,130.886,-50.932,-178.233,5.809,148.503
C09937=1216.682,130.637,-50.911,-178.236,5.809,148.503
C09938=1216.687,130.389,-50.891,-178.238,5.807,148.504
C09939=1216.691,130.139,-50.872,-178.241,5.806,148.504
C09940=1216.696,129.890,-50.851,-178.244,5.804,148.505
C09941=1216.700,129.641,-50.832,-178.246,5.804,148.505
C09942=1216.706,129.391,-50.811,-178.248,5.803,148.506
C09943=1216.710,129.143,-50.790,-178.252,5.801,148.506
C09944=1216.715,128.893,-50.771,-178.254,5.800,148.507
C09945=1216.720,128.645,-50.751,-178.257,5.799,148.507
C09946=1216.725,128.395,-50.731,-178.259,5.798,148.508
C09947=1216.729,128.146,-50.711,-178.262,5.797,148.508
C09948=1216.734,127.897,-50.691,-178.264,5.796,148.509
C09949=1216.738,127.648,-50.670,-178.266,5.795,148.509
C09950=1216.744,127.399,-50.651,-178.270,5.793,148.510
C09951=1216.748,127.150,-50.631,-178.272,5.792,148.510
C09952=1216.753,126.900,-50.611,-178.275,5.791,148.511
C09953=1216.758,126.651,-50.590,-178.277,5.790,148.511
C09954=1216.763,126.401,-50.571,-178.280,5.789,148.512
C09955=1216.768,126.153,-50.551,-178.282,5.787,148.512
C09956=1216.772,125.904,-50.531,-178.285,5.787,148.513
C09957=1216.777,125.655,-50.511,-178.288,5.785,148.513
C09958=1216.782,125.405,-50.491,-178.290,5.784,148.514
C09959=1216.786,125.156,-50.471,-178.292,5.783,148.514
C09960=1216.791,124.907,-50.451,-178.295,5.782,148.515
C09961=1216.796,124.658,-50.432,-178.298,5.781,148.515
C09962=1216.801,124.409,-50.411,-178.301,5.780,148.516
C09963=1216.805,124.159,-50.392,-178.303,5.779,148.516
C09964=1216.811,123.910,-50.372,-178.305,5.778,148.517
C09965=1216.815,123.661,-50.352,-178.308,5.776,148.517
C09966=1216.820,123.412,-50.332,-178.311,5.776,148.518
C09967=1216.825,123.162,-50.313,-178.313,5.774,148.518
C09968=1216.830,122.914,-50.293,-178.316,5.773,148.519
C09969=1216.834,122.664,-50.273,-178.318,5.772,148.520
C09970=1216.839,122.415,-50.253,-178.321,5.771,148.520
C09971=1216.844,122.166,-50.233,-178.323,5.770,148.521
C09972=1216.849,121.917,-50.214,-178.326,5.769,148.521
C09973=1216.854,121.667,-50.194,-178.329,5.767,148.522
C09974=1216.858,121.418,-50.175,-178.331,5.767,148.522
C09975=1216.862,121.169,-50.154,-178.334,5.765,148.523
C09976=1216.867,120.920,-50.135,-178.337,5.764,148.523
C09977=1216.872,120.671,-50.116,-178.339,5.763,148.524
C09978=1216.877,120.421,-50.096,-178.342,5.762,148.524
C09979=1216.882,120.173,-50.076,-178.344,5.761,148.525
C09980=1216.887,119.923,-50.056,-178.347,5.760,148.525
C09981=1216.891,119.674,-50.037,-178.349,5.759,148.526
C09982=1216.897,119.425,-50.017,-178.352,5.758,148.526
C09983=1216.901,119.176,-49.997,-178.355,5.756,148.527
C09984=1216.905,118.927,-49.978,-178.357,5.756,148.527
C09985=1216.911,118.678,-49.959,-178.359,5.755,148.528
C09986=1216.915,118.428,-49.939,-178.363,5.753,148.528
C09987=1216.920,118.179,-49.919,-178.365,5.752,148.529
C09988=1216.925,117.930,-49.900,-178.367,5.752,148.529
C09989=1216.930,117.680,-49.880,-178.370,5.750,148.530
C09990=1216.935,117.431,-49.860,-178.373,5.749,148.531
C09991=1216.939,117.183,-49.841,-178.375,5.748,148.531
C09992=1216.944,116.933,-49.822,-178.378,5.747,148.532
C09993=1216.949,116.684,-49.802,-178.380,5.746,148.532
C09994=1216.954,116.435,-49.783,-178.383,5.745,148.533
C09995=1216.959,116.185,-49.763,-178.386,5.744,148.533
C09996=1216.963,115.937,-49.744,-178.388,5.743,148.534
//INST
///DATE 2021/06/25 14:27
///ATTR SC,RW,RJ
////FRAME ROBOT
///GROUP1 RB1
NOP
MOVL C00000 V=800.0 PL=0
MOVL C00001 V=800.0 PL=0
MOVL C00002 V=800.0 PL=0
MOVL C00003 V=800.0 PL=0
MOVL C00004 V=800.0 PL=0
MOVL C00005 V=800.0 PL=0
MOVL C00006 V=800.0 PL=0
MOVL C00007 V=800.0 PL=0
MOVL C00008 V=800.0 PL=0
MOVL C00009 V=800.0 PL=0
MOVL C00010 V=800.0 PL=0
MOVL C00011 V=800.0 PL=0
MOVL C00012 V=800.0 PL=0
MOVL C00013 V=800.0 PL=0
MOVL C00014 V=800.0 PL=0
MOVL C00015 V=800.0 PL=0
MOVL C00016 V=800.0 PL=0
MOVL C00017 V=800.0 PL=0
MOVL C00018 V=800.0 PL=0
MOVL C00019 V=800.0 PL=0
MOVL C00020 V=800.0 PL=0
MOVL C00021 V=800.0 PL=0
MOVL C00022 V=800.0 PL=0
MOVL C00023 V=800.0 PL=0
MOVL C00024 V=800.0 PL=0
MOVL C00025 V=800.0 PL=0
MOVL C00026 V=800.0 PL=0
MOVL C00027 V=800.0 PL=0
MOVL C00028 V=800.0 PL=0
MOVL C00029 V=800.0 PL=0
MOVL C00030 V=800.0 PL=0
MOVL C00031 V=800.0 PL=0
MOVL C00032 V=800.0 PL=0
MOVL C00033 V=800.0 PL=0
MOVL C00034 V=800.0 PL=0
MOVL C00035 V=800.0 PL=0
MOVL C00036 V=800.0 PL=0
MOVL C00037 V=800.0 PL=0
MOVL C00038 V=800.0 PL=0
MOVL C00039 V=800.0 PL=0
MOVL C00040 V=800.0 PL=0
MOVL C00041 V=800.0 PL=0
MOVL C00042 V=800.0 PL=0
MOVL C00043 V=800.0 PL=0
MOVL C00044 V=800.0 PL=0
MOVL C00045 V=800.0 PL=0
MOVL C00046 V=800.0 PL=0
MOVL C00047 V=800.0 PL=0
MOVL C00048 V=800.0 PL=0
MOVL C00049 V=800.0 PL=0
MOVL C00050 V=800.0 PL=0
MOVL C00051 V=800.0 PL=0
MOVL C00052 V=800.0 PL=0
MOVL C00053 V=800.0 PL=0
MOVL C00054 V=800.0 PL=0
MOVL C00055 V=800.0 PL=0
MOVL C00056 V=800.0 PL=0
MOVL C00057 V=800.0 PL=0
MOVL C00058 V=800.0 PL=0
MOVL C00059 V=800.0 PL=0
MOVL C00060 V=800.0 PL=0
MOVL C00061 V=800.0 PL=0
MOVL C00062 V=800.0 PL=0
MOVL C00063 V=800.0 PL=0
MOVL C00064 V=800.0 PL=0
MOVL C00065 V=800.0 PL=0
MOVL C00066 V=800.0 PL=0
MOVL C00067 V=800.0 PL=0
MOVL C00068 V=800.0 PL=0
MOVL C00069 V=800.0 PL=0
MOVL C00070 V=800.0 PL=0
MOVL C00071 V=800.0 PL=0
MOVL C00072 V=800.0 PL=0
MOVL C00073 V=800.0 PL=0
MOVL C00074 V=800.0 PL=0
MOVL C00075 V=800.0 PL=0
MOVL C00076 V=800.0 PL=0
MOVL C00077 V=800.0 PL=0
MOVL C00078 V=800.0 PL=0
MOVL C00079 V=800.0 PL=0
MOVL C00080 V=800.0 PL=0
MOVL C00081 V=800.0 PL=0
MOVL C00082 V=800.0 PL=0
MOVL C00083 V=800.0 PL=0
MOVL C00084 V=800.0 PL=0
MOVL C00085 V=800.0 PL=0
MOVL C00086 V=800.0 PL=0
MOVL C00087 V=800.0 PL=0
MOVL C00088 V=800.0 PL=0
MOVL C00089 V=800.0 PL=0
MOVL C00090 V=800.0 PL=0
MOVL C00091 V=800.0 PL=0
MOVL C00092 V=800.0 PL=0
MOVL C00093 V=800.0 PL=0
MOVL C00094 V=800.0 PL=0
MOVL C00095 V=800.0 PL=0
MOVL C00096 V=800.0 PL=0
MOVL C00097 V=800.0 PL=0
MOVL C00098 V=800.0 PL=0
MOVL C00099 V=800.0 PL=0
MOVL C00100 V=800.0 PL=0
MOVL C00101 V=800.0 PL=0
MOVL C00102 V=800.0 PL=0
MOVL C00103 V=800.0 PL=0
MOVL C00104 V=800.0 PL=0
MOVL C00105 V=800.0 PL=0
MOVL C00106 V=800.0 PL=0
MOVL C00107 V=800.0 PL=0
MOVL C00108 V=800.0 PL=0
MOVL C00109 V=800.0 PL=0
MOVL C00110 V=800.0 PL=0
MOVL C00111 V=800.0 PL=0
MOVL C00112 V=800.0 PL=0
MOVL C00113 V=800.0 PL=0
MOVL C00114 V=800.0 PL=0
MOVL C00115 V=800.0 PL=0
MOVL C00116 V=800.0 PL=0
MOVL C00117 V=800.0 PL=0
MOVL C00118 V=800.0 PL=0
MOVL C00119 V=800.0 PL=0
MOVL C00120 V=800.0 PL=0
MOVL C00121 V=800.0 PL=0
MOVL C00122 V=800.0 PL=0
MOVL C00123 V=800.0 PL=0
MOVL C00124 V=800.0 PL=0
MOVL C00125 V=800.0 PL=0
MOVL C00126 V=800.0 PL=0
MOVL C00127 V=800.0 PL=0
MOVL C00128 V=800.0 PL=0
MOVL C00129 V=800.0 PL=0
MOVL C00130 V=800.0 PL=0
MOVL C00131 V=800.0 PL=0
MOVL C00132 V=800.0 PL=0
MOVL C00133 V=800.0 PL=0
MOVL C00134 V=800.0 PL=0
MOVL C00135 V=800.0 PL=0
MOVL C00136 V=800.0 PL=0
MOVL C00137 V=800.0 PL=0
MOVL C00138 V=800.0 PL=0
MOVL C00139 V=800.0 PL=0
MOVL C00140 V=800.0 PL=0
MOVL C00141 V=800.0 PL=0
MOVL C00142 V=800.0 PL=0
MOVL C00143 V=800.0 PL=0
MOVL C00144 V=800.0 PL=0
MOVL C00145 V=800.0 PL=0
MOVL C00146 V=800.0 PL=0
MOVL C00147 V=800.0 PL=0
MOVL C00148 V=800.0 PL=0
MOVL C00149 V=800.0 PL=0
MOVL C00150 V=800.0 PL=0
MOVL C00151 V=800.0 PL=0
MOVL C00152 V=800.0 PL=0
MOVL C00153 V=800.0 PL=0
MOVL C00154 V=800.0 PL=0
MOVL C00155 V=800.0 PL=0
MOVL C00156 V=800.0 PL=0
MOVL C00157 V=800.0 PL=0
MOVL C00158 V=800.0 PL=0
MOVL C00159 V=800.0 PL=0
MOVL C00160 V=800.0 PL=0
MOVL C00161 V=800.0 PL=0
MOVL C00162 V=800.0 PL=0
MOVL C00163 V=800.0 PL=0
MOVL C00164 V=800.0 PL=0
MOVL C00165 V=800.0 PL=0
MOVL C00166 V=800.0 PL=0
MOVL C00167 V=800.0 PL=0
MOVL C00168 V=800.0 PL=0
MOVL C00169 V=800.0 PL=0
MOVL C00170 V=800.0 PL=0
MOVL C00171 V=800.0 PL=0
MOVL C00172 V=800.0 PL=0
MOVL C00173 V=800.0 PL=0
MOVL C00174 V=800.0 PL=0
MOVL C00175 V=800.0 PL=0
MOVL C00176 V=800.0 PL=0
MOVL C00177 V=800.0 PL=0
MOVL C00178 V=800.0 PL=0
MOVL C00179 V=800.0 PL=0
MOVL C00180 V=800.0 PL=0
MOVL C00181 V=800.0 PL=0
MOVL C00182 V=800.0 PL=0
MOVL C00183 V=800.0 PL=0
MOVL C00184 V=800.0 PL=0
MOVL C00185 V=800.0 PL=0
MOVL C00186 V=800.0 PL=0
MOVL C00187 V=800.0 PL=0
MOVL C00188 V=800.0 PL=0
MOVL C00189 V=800.0 PL=0
MOVL C00190 V=800.0 PL=0
MOVL C00191 V=800.0 PL=0
MOVL C00192 V=800.0 PL=0
MOVL C00193 V=800.0 PL=0
MOVL C00194 V=800.0 PL=0
MOVL C00195 V=800.0 PL=0
MOVL C00196 V=800.0 PL=0
MOVL C00197 V=800.0 PL=0
MOVL C00198 V=800.0 PL=0
MOVL C00199 V=800.0 PL=0
MOVL C00200 V=800.0 PL=0
MOVL C00201 V=800.0 PL=0
MOVL C00202 V=800.0 PL=0
MOVL C00203 V=800.0 PL=0
MOVL C00204 V=800.0 PL=0
MOVL C00205 V=800.0 PL=0
MOVL C00206 V=800.0 PL=0
MOVL C00207 V=800.0 PL=0
MOVL C00208 V=800.0 PL=0
MOVL C00209 V=800.0 PL=0
MOVL C00210 V=800.0 PL=0
MOVL C00211 V=800.0 PL=0
MOVL C00212 V=800.0 PL=0
MOVL C00213 V=800.0 PL=0
MOVL C00214 V=800.0 PL=0
MOVL C00215 V=800.0 PL=0
MOVL C00216 V=800.0 PL=0
MOVL C00217 V=800.0 PL=0
MOVL C00218 V=800.0 PL=0
MOVL C00219 V=800.0 PL=0
MOVL C00220 V=800.0 PL=0
MOVL C00221 V=800.0 PL=0
MOVL C00222 V=800.0 PL=0
MOVL C00223 V=800.0 PL=0
MOVL C00224 V=800.0 PL=0
MOVL C00225 V=800.0 PL=0
MOVL C00226 V=800.0 PL=0
MOVL C00227 V=800.0 PL=0
MOVL C00228 V=800.0 PL=0
MOVL C00229 V=800.0 PL=0
MOVL C00230 V=800.0 PL=0
MOVL C00231 V=800.0 PL=0
MOVL C00232 V=800.0 PL=0
MOVL C00233 V=800.0 PL=0
MOVL C00234 V=800.0 PL=0
MOVL C00235 V=800.0 PL=0
MOVL C00236 V=800.0 PL=0
MOVL C00237 V=800.0 PL=0
MOVL C00238 V=800.0 PL=0
MOVL C00239 V=800.0 PL=0
MOVL C00240 V=800.0 PL=0
MOVL C00241 V=800.0 PL=0
MOVL C00242 V=800.0 PL=0
MOVL C00243 V=800.0 PL=0
MOVL C00244 V=800.0 PL=0
MOVL C00245 V=800.0 PL=0
MOVL C00246 V=800.0 PL=0
MOVL C00247 V=800.0 PL=0
MOVL C00248 V=800.0 PL=0
MOVL C00249 V=800.0 PL=0
MOVL C00250 V=800.0 PL=0
MOVL C00251 V=800.0 PL=0
MOVL C00252 V=800.0 PL=0
MOVL C00253 V=800.0 PL=0
MOVL C00254 V=800.0 PL=0
MOVL C00255 V=800.0 PL=0
MOVL C00256 V=800.0 PL=0
MOVL C00257 V=800.0 PL=0
MOVL C00258 V=800.0 PL=0
MOVL C00259 V=800.0 PL=0
MOVL C00260 V=800.0 PL=0
MOVL C00261 V=800.0 PL=0
MOVL C00262 V=800.0 PL=0
MOVL C00263 V=800.0 PL=0
MOVL C00264 V=800.0 PL=0
MOVL C00265 V=800.0 PL=0
MOVL C00266 V=800.0 PL=0
MOVL C00267 V=800.0 PL=0
MOVL C00268 V=800.0 PL=0
MOVL C00269 V=800.0 PL=0
MOVL C00270 V=800.0 PL=0
MOVL C00271 V=800.0 PL=0
MOVL C00272 V=800.0 PL=0
MOVL C00273 V=800.0 PL=0
MOVL C00274 V=800.0 PL=0
MOVL C00275 V=800.0 PL=0
MOVL C00276 V=800.0 PL=0
MOVL C00277 V=800.0 PL=0
MOVL C00278 V=800.0 PL=0
MOVL C00279 V=800.0 PL=0
MOVL C00280 V=800.0 PL=0
MOVL C00281 V=800.0 PL=0
MOVL C00282 V=800.0 PL=0
MOVL C00283 V=800.0 PL=0
MOVL C00284 V=800.0 PL=0
MOVL C00285 V=800.0 PL=0
MOVL C00286 V=800.0 PL=0
MOVL C00287 V=800.0 PL=0
MOVL C00288 V=800.0 PL=0
MOVL C00289 V=800.0 PL=0
MOVL C00290 V=800.0 PL=0
MOVL C00291 V=800.0 PL=0
MOVL C00292 V=800.0 PL=0
MOVL C00293 V=800.0 PL=0
MOVL C00294 V=800.0 PL=0
MOVL C00295 V=800.0 PL=0
MOVL C00296 V=800.0 PL=0
MOVL C00297 V=800.0 PL=0
MOVL C00298 V=800.0 PL=0
MOVL C00299 V=800.0 PL=0
MOVL C00300 V=800.0 PL=0
MOVL C00301 V=800.0 PL=0
MOVL C00302 V=800.0 PL=0
MOVL C00303 V=800.0 PL=0
MOVL C00304 V=800.0 PL=0
MOVL C00305 V=800.0 PL=0
MOVL C00306 V=800.0 PL=0
MOVL C00307 V=800.0 PL=0
MOVL C00308 V=800.0 PL=0
MOVL C00309 V=800.0 PL=0
MOVL C00310 V=800.0 PL=0
MOVL C00311 V=800.0 PL=0
MOVL C00312 V=800.0 PL=0
MOVL C00313 V=800.0 PL=0
MOVL C00314 V=800.0 PL=0
MOVL C00315 V=800.0 PL=0
MOVL C00316 V=800.0 PL=0
MOVL C00317 V=800.0 PL=0
MOVL C00318 V=800.0 PL=0
MOVL C00319 V=800.0 PL=0
MOVL C00320 V=800.0 PL=0
MOVL C00321 V=800.0 PL=0
MOVL C00322 V=800.0 PL=0
MOVL C00323 V=800.0 PL=0
MOVL C00324 V=800.0 PL=0
MOVL C00325 V=800.0 PL=0
MOVL C00326 V=800.0 PL=0
MOVL C00327 V=800.0 PL=0
MOVL C00328 V=800.0 PL=0
MOVL C00329 V=800.0 PL=0
MOVL C00330 V=800.0 PL=0
MOVL C00331 V=800.0 PL=0
MOVL C00332 V=800.0 PL=0
MOVL C00333 V=800.0 PL=0
MOVL C00334 V=800.0 PL=0
MOVL C00335 V=800.0 PL=0
MOVL C00336 V=800.0 PL=0
MOVL C00337 V=800.0 PL=0
MOVL C00338 V=800.0 PL=0
MOVL C00339 V=800.0 PL=0
MOVL C00340 V=800.0 PL=0
MOVL C00341 V=800.0 PL=0
MOVL C00342 V=800.0 PL=0
MOVL C00343 V=800.0 PL=0
MOVL C00344 V=800.0 PL=0
MOVL C00345 V=800.0 PL=0
MOVL C00346 V=800.0 PL=0
MOVL C00347 V=800.0 PL=0
MOVL C00348 V=800.0 PL=0
MOVL C00349 V=800.0 PL=0
MOVL C00350 V=800.0 PL=0
MOVL C00351 V=800.0 PL=0
MOVL C00352 V=800.0 PL=0
MOVL C00353 V=800.0 PL=0
MOVL C00354 V=800.0 PL=0
MOVL C00355 V=800.0 PL=0
MOVL C00356 V=800.0 PL=0
MOVL C00357 V=800.0 PL=0
MOVL C00358 V=800.0 PL=0
MOVL C00359 V=800.0 PL=0
MOVL C00360 V=800.0 PL=0
MOVL C00361 V=800.0 PL=0
MOVL C00362 V=800.0 PL=0
MOVL C00363 V=800.0 PL=0
MOVL C00364 V=800.0 PL=0
MOVL C00365 V=800.0 PL=0
MOVL C00366 V=800.0 PL=0
MOVL C00367 V=800.0 PL=0
MOVL C00368 V=800.0 PL=0
MOVL C00369 V=800.0 PL=0
MOVL C00370 V=800.0 PL=0
MOVL C00371 V=800.0 PL=0
MOVL C00372 V=800.0 PL=0
MOVL C00373 V=800.0 PL=0
MOVL C00374 V=800.0 PL=0
MOVL C00375 V=800.0 PL=0
MOVL C00376 V=800.0 PL=0
MOVL C00377 V=800.0 PL=0
MOVL C00378 V=800.0 PL=0
MOVL C00379 V=800.0 PL=0
MOVL C00380 V=800.0 PL=0
MOVL C00381 V=800.0 PL=0
MOVL C00382 V=800.0 PL=0
MOVL C00383 V=800.0 PL=0
MOVL C00384 V=800.0 PL=0
MOVL C00385 V=800.0 PL=0
MOVL C00386 V=800.0 PL=0
MOVL C00387 V=800.0 PL=0
MOVL C00388 V=800.0 PL=0
MOVL C00389 V=800.0 PL=0
MOVL C00390 V=800.0 PL=0
MOVL C00391 V=800.0 PL=0
MOVL C00392 V=800.0 PL=0
MOVL C00393 V=800.0 PL=0
MOVL C00394 V=800.0 PL=0
MOVL C00395 V=800.0 PL=0
MOVL C00396 V=800.0 PL=0
MOVL C00397 V=800.0 PL=0
MOVL C00398 V=800.0 PL=0
MOVL C00399 V=800.0 PL=0
MOVL C00400 V=800.0 PL=0
MOVL C00401 V=800.0 PL=0
MOVL C00402 V=800.0 PL=0
MOVL C00403 V=800.0 PL=0
MOVL C00404 V=800.0 PL=0
MOVL C00405 V=800.0 PL=0
MOVL C00406 V=800.0 PL=0
MOVL C00407 V=800.0 PL=0
MOVL C00408 V=800.0 PL=0
MOVL C00409 V=800.0 PL=0
MOVL C00410 V=800.0 PL=0
MOVL C00411 V=800.0 PL=0
MOVL C00412 V=800.0 PL=0
MOVL C00413 V=800.0 PL=0
MOVL C00414 V=800.0 PL=0
MOVL C00415 V=800.0 PL=0
MOVL C00416 V=800.0 PL=0
MOVL C00417 V=800.0 PL=0
MOVL C00418 V=800.0 PL=0
MOVL C00419 V=800.0 PL=0
MOVL C00420 V=800.0 PL=0
MOVL C00421 V=800.0 PL=0
MOVL C00422 V=800.0 PL=0
MOVL C00423 V=800.0 PL=0
MOVL C00424 V=800.0 PL=0
MOVL C00425 V=800.0 PL=0
MOVL C00426 V=800.0 PL=0
MOVL C00427 V=800.0 PL=0
MOVL C00428 V=800.0 PL=0
MOVL C00429 V=800.0 PL=0
MOVL C00430 V=800.0 PL=0
MOVL C00431 V=800.0 PL=0
MOVL C00432 V=800.0 PL=0
MOVL C00433 V=800.0 PL=0
MOVL C00434 V=800.0 PL=0
MOVL C00435 V=800.0 PL=0
MOVL C00436 V=800.0 PL=0
MOVL C00437 V=800.0 PL=0
MOVL C00438 V=800.0 PL=0
MOVL C00439 V=800.0 PL=0
MOVL C00440 V=800.0 PL=0
MOVL C00441 V=800.0 PL=0
MOVL C00442 V=800.0 PL=0
MOVL C00443 V=800.0 PL=0
MOVL C00444 V=800.0 PL=0
MOVL C00445 V=800.0 PL=0
MOVL C00446 V=800.0 PL=0
MOVL C00447 V=800.0 PL=0
MOVL C00448 V=800.0 PL=0
MOVL C00449 V=800.0 PL=0
MOVL C00450 V=800.0 PL=0
MOVL C00451 V=800.0 PL=0
MOVL C00452 V=800.0 PL=0
MOVL C00453 V=800.0 PL=0
MOVL C00454 V=800.0 PL=0
MOVL C00455 V=800.0 PL=0
MOVL C00456 V=800.0 PL=0
MOVL C00457 V=800.0 PL=0
MOVL C00458 V=800.0 PL=0
MOVL C00459 V=800.0 PL=0
MOVL C00460 V=800.0 PL=0
MOVL C00461 V=800.0 PL=0
MOVL C00462 V=800.0 PL=0
MOVL C00463 V=800.0 PL=0
MOVL C00464 V=800.0 PL=0
MOVL C00465 V=800.0 PL=0
MOVL C00466 V=800.0 PL=0
MOVL C00467 V=800.0 PL=0
MOVL C00468 V=800.0 PL=0
MOVL C00469 V=800.0 PL=0
MOVL C00470 V=800.0 PL=0
MOVL C00471 V=800.0 PL=0
MOVL C00472 V=800.0 PL=0
MOVL C00473 V=800.0 PL=0
MOVL C00474 V=800.0 PL=0
MOVL C00475 V=800.0 PL=0
MOVL C00476 V=800.0 PL=0
MOVL C00477 V=800.0 PL=0
MOVL C00478 V=800.0 PL=0
MOVL C00479 V=800.0 PL=0
MOVL C00480 V=800.0 PL=0
MOVL C00481 V=800.0 PL=0
MOVL C00482 V=800.0 PL=0
MOVL C00483 V=800.0 PL=0
MOVL C00484 V=800.0 PL=0
MOVL C00485 V=800.0 PL=0
MOVL C00486 V=800.0 PL=0
MOVL C00487 V=800.0 PL=0
MOVL C00488 V=800.0 PL=0
MOVL C00489 V=800.0 PL=0
MOVL C00490 V=800.0 PL=0
MOVL C00491 V=800.0 PL=0
MOVL C00492 V=800.0 PL=0
MOVL C00493 V=800.0 PL=0
MOVL C00494 V=800.0 PL=0
MOVL C00495 V=800.0 PL=0
MOVL C00496 V=800.0 PL=0
MOVL C00497 V=800.0 PL=0
MOVL C00498 V=800.0 PL=0
MOVL C00499 V=800.0 PL=0
MOVL C00500 V=800.0 PL=0
MOVL C00501 V=800.0 PL=0
MOVL C00502 V=800.0 PL=0
MOVL C00503 V=800.0 PL=0
MOVL C00504 V=800.0 PL=0
MOVL C00505 V=800.0 PL=0
MOVL C00506 V=800.0 PL=0
MOVL C00507 V=800.0 PL=0
MOVL C00508 V=800.0 PL=0
MOVL C00509 V=800.0 PL=0
MOVL C00510 V=800.0 PL=0
MOVL C00511 V=800.0 PL=0
MOVL C00512 V=800.0 PL=0
MOVL C00513 V=800.0 PL=0
MOVL C00514 V=800.0 PL=0
MOVL C00515 V=800.0 PL=0
MOVL C00516 V=800.0 PL=0
MOVL C00517 V=800.0 PL=0
MOVL C00518 V=800.0 PL=0
MOVL C00519 V=800.0 PL=0
MOVL C00520 V=800.0 PL=0
MOVL C00521 V=800.0 PL=0
MOVL C00522 V=800.0 PL=0
MOVL C00523 V=800.0 PL=0
MOVL C00524 V=800.0 PL=0
MOVL C00525 V=800.0 PL=0
MOVL C00526 V=800.0 PL=0
MOVL C00527 V=800.0 PL=0
MOVL C00528 V=800.0 PL=0
MOVL C00529 V=800.0 PL=0
MOVL C00530 V=800.0 PL=0
MOVL C00531 V=800.0 PL=0
MOVL C00532 V=800.0 PL=0
MOVL C00533 V=800.0 PL=0
MOVL C00534 V=800.0 PL=0
MOVL C00535 V=800.0 PL=0
MOVL C00536 V=800.0 PL=0
MOVL C00537 V=800.0 PL=0
MOVL C00538 V=800.0 PL=0
MOVL C00539 V=800.0 PL=0
MOVL C00540 V=800.0 PL=0
MOVL C00541 V=800.0 PL=0
MOVL C00542 V=800.0 PL=0
MOVL C00543 V=800.0 PL=0
MOVL C00544 V=800.0 PL=0
MOVL C00545 V=800.0 PL=0
MOVL C00546 V=800.0 PL=0
MOVL C00547 V=800.0 PL=0
MOVL C00548 V=800.0 PL=0
MOVL C00549 V=800.0 PL=0
MOVL C00550 V=800.0 PL=0
MOVL C00551 V=800.0 PL=0
MOVL C00552 V=800.0 PL=0
MOVL C00553 V=800.0 PL=0
MOVL C00554 V=800.0 PL=0
MOVL C00555 V=800.0 PL=0
MOVL C00556 V=800.0 PL=0
MOVL C00557 V=800.0 PL=0
MOVL C00558 V=800.0 PL=0
MOVL C00559 V=800.0 PL=0
MOVL C00560 V=800.0 PL=0
MOVL C00561 V=800.0 PL=0
MOVL C00562 V=800.0 PL=0
MOVL C00563 V=800.0 PL=0
MOVL C00564 V=800.0 PL=0
MOVL C00565 V=800.0 PL=0
MOVL C00566 V=800.0 PL=0
MOVL C00567 V=800.0 PL=0
MOVL C00568 V=800.0 PL=0
MOVL C00569 V=800.0 PL=0
MOVL C00570 V=800.0 PL=0
MOVL C00571 V=800.0 PL=0
MOVL C00572 V=800.0 PL=0
MOVL C00573 V=800.0 PL=0
MOVL C00574 V=800.0 PL=0
MOVL C00575 V=800.0 PL=0
MOVL C00576 V=800.0 PL=0
MOVL C00577 V=800.0 PL=0
MOVL C00578 V=800.0 PL=0
MOVL C00579 V=800.0 PL=0
MOVL C00580 V=800.0 PL=0
MOVL C00581 V=800.0 PL=0
MOVL C00582 V=800.0 PL=0
MOVL C00583 V=800.0 PL=0
MOVL C00584 V=800.0 PL=0
MOVL C00585 V=800.0 PL=0
MOVL C00586 V=800.0 PL=0
MOVL C00587 V=800.0 PL=0
MOVL C00588 V=800.0 PL=0
MOVL C00589 V=800.0 PL=0
MOVL C00590 V=800.0 PL=0
MOVL C00591 V=800.0 PL=0
MOVL C00592 V=800.0 PL=0
MOVL C00593 V=800.0 PL=0
MOVL C00594 V=800.0 PL=0
MOVL C00595 V=800.0 PL=0
MOVL C00596 V=800.0 PL=0
MOVL C00597 V=800.0 PL=0
MOVL C00598 V=800.0 PL=0
MOVL C00599 V=800.0 PL=0
MOVL C00600 V=800.0 PL=0
MOVL C00601 V=800.0 PL=0
MOVL C00602 V=800.0 PL=0
MOVL C00603 V=800.0 PL=0
MOVL C00604 V=800.0 PL=0
MOVL C00605 V=800.0 PL=0
MOVL C00606 V=800.0 PL=0
MOVL C00607 V=800.0 PL=0
MOVL C00608 V=800.0 PL=0
MOVL C00609 V=800.0 PL=0
MOVL C00610 V=800.0 PL=0
MOVL C00611 V=800.0 PL=0
MOVL C00612 V=800.0 PL=0
MOVL C00613 V=800.0 PL=0
MOVL C00614 V=800.0 PL=0
MOVL C00615 V=800.0 PL=0
MOVL C00616 V=800.0 PL=0
MOVL C00617 V=800.0 PL=0
MOVL C00618 V=800.0 PL=0
MOVL C00619 V=800.0 PL=0
MOVL C00620 V=800.0 PL=0
MOVL C00621 V=800.0 PL=0
MOVL C00622 V=800.0 PL=0
MOVL C00623 V=800.0 PL=0
MOVL C00624 V=800.0 PL=0
MOVL C00625 V=800.0 PL=0
MOVL C00626 V=800.0 PL=0
MOVL C00627 V=800.0 PL=0
MOVL C00628 V=800.0 PL=0
MOVL C00629 V=800.0 PL=0
MOVL C00630 V=800.0 PL=0
MOVL C00631 V=800.0 PL=0
MOVL C00632 V=800.0 PL=0
MOVL C00633 V=800.0 PL=0
MOVL C00634 V=800.0 PL=0
MOVL C00635 V=800.0 PL=0
MOVL C00636 V=800.0 PL=0
MOVL C00637 V=800.0 PL=0
MOVL C00638 V=800.0 PL=0
MOVL C00639 V=800.0 PL=0
MOVL C00640 V=800.0 PL=0
MOVL C00641 V=800.0 PL=0
MOVL C00642 V=800.0 PL=0
MOVL C00643 V=800.0 PL=0
MOVL C00644 V=800.0 PL=0
MOVL C00645 V=800.0 PL=0
MOVL C00646 V=800.0 PL=0
MOVL C00647 V=800.0 PL=0
MOVL C00648 V=800.0 PL=0
MOVL C00649 V=800.0 PL=0
MOVL C00650 V=800.0 PL=0
MOVL C00651 V=800.0 PL=0
MOVL C00652 V=800.0 PL=0
MOVL C00653 V=800.0 PL=0
MOVL C00654 V=800.0 PL=0
MOVL C00655 V=800.0 PL=0
MOVL C00656 V=800.0 PL=0
MOVL C00657 V=800.0 PL=0
MOVL C00658 V=800.0 PL=0
MOVL C00659 V=800.0 PL=0
MOVL C00660 V=800.0 PL=0
MOVL C00661 V=800.0 PL=0
MOVL C00662 V=800.0 PL=0
MOVL C00663 V=800.0 PL=0
MOVL C00664 V=800.0 PL=0
MOVL C00665 V=800.0 PL=0
MOVL C00666 V=800.0 PL=0
MOVL C00667 V=800.0 PL=0
MOVL C00668 V=800.0 PL=0
MOVL C00669 V=800.0 PL=0
MOVL C00670 V=800.0 PL=0
MOVL C00671 V=800.0 PL=0
MOVL C00672 V=800.0 PL=0
MOVL C00673 V=800.0 PL=0
MOVL C00674 V=800.0 PL=0
MOVL C00675 V=800.0 PL=0
MOVL C00676 V=800.0 PL=0
MOVL C00677 V=800.0 PL=0
MOVL C00678 V=800.0 PL=0
MOVL C00679 V=800.0 PL=0
MOVL C00680 V=800.0 PL=0
MOVL C00681 V=800.0 PL=0
MOVL C00682 V=800.0 PL=0
MOVL C00683 V=800.0 PL=0
MOVL C00684 V=800.0 PL=0
MOVL C00685 V=800.0 PL=0
MOVL C00686 V=800.0 PL=0
MOVL C00687 V=800.0 PL=0
MOVL C00688 V=800.0 PL=0
MOVL C00689 V=800.0 PL=0
MOVL C00690 V=800.0 PL=0
MOVL C00691 V=800.0 PL=0
MOVL C00692 V=800.0 PL=0
MOVL C00693 V=800.0 PL=0
MOVL C00694 V=800.0 PL=0
MOVL C00695 V=800.0 PL=0
MOVL C00696 V=800.0 PL=0
MOVL C00697 V=800.0 PL=0
MOVL C00698 V=800.0 PL=0
MOVL C00699 V=800.0 PL=0
MOVL C00700 V=800.0 PL=0
MOVL C00701 V=800.0 PL=0
MOVL C00702 V=800.0 PL=0
MOVL C00703 V=800.0 PL=0
MOVL C00704 V=800.0 PL=0
MOVL C00705 V=800.0 PL=0
MOVL C00706 V=800.0 PL=0
MOVL C00707 V=800.0 PL=0
MOVL C00708 V=800.0 PL=0
MOVL C00709 V=800.0 PL=0
MOVL C00710 V=800.0 PL=0
MOVL C00711 V=800.0 PL=0
MOVL C00712 V=800.0 PL=0
MOVL C00713 V=800.0 PL=0
MOVL C00714 V=800.0 PL=0
MOVL C00715 V=800.0 PL=0
MOVL C00716 V=800.0 PL=0
MOVL C00717 V=800.0 PL=0
MOVL C00718 V=800.0 PL=0
MOVL C00719 V=800.0 PL=0
MOVL C00720 V=800.0 PL=0
MOVL C00721 V=800.0 PL=0
MOVL C00722 V=800.0 PL=0
MOVL C00723 V=800.0 PL=0
MOVL C00724 V=800.0 PL=0
MOVL C00725 V=800.0 PL=0
MOVL C00726 V=800.0 PL=0
MOVL C00727 V=800.0 PL=0
MOVL C00728 V=800.0 PL=0
MOVL C00729 V=800.0 PL=0
MOVL C00730 V=800.0 PL=0
MOVL C00731 V=800.0 PL=0
MOVL C00732 V=800.0 PL=0
MOVL C00733 V=800.0 PL=0
MOVL C00734 V=800.0 PL=0
MOVL C00735 V=800.0 PL=0
MOVL C00736 V=800.0 PL=0
MOVL C00737 V=800.0 PL=0
MOVL C00738 V=800.0 PL=0
MOVL C00739 V=800.0 PL=0
MOVL C00740 V=800.0 PL=0
MOVL C00741 V=800.0 PL=0
MOVL C00742 V=800.0 PL=0
MOVL C00743 V=800.0 PL=0
MOVL C00744 V=800.0 PL=0
MOVL C00745 V=800.0 PL=0
MOVL C00746 V=800.0 PL=0
MOVL C00747 V=800.0 PL=0
MOVL C00748 V=800.0 PL=0
MOVL C00749 V=800.0 PL=0
MOVL C00750 V=800.0 PL=0
MOVL C00751 V=800.0 PL=0
MOVL C00752 V=800.0 PL=0
MOVL C00753 V=800.0 PL=0
MOVL C00754 V=800.0 PL=0
MOVL C00755 V=800.0 PL=0
MOVL C00756 V=800.0 PL=0
MOVL C00757 V=800.0 PL=0
MOVL C00758 V=800.0 PL=0
MOVL C00759 V=800.0 PL=0
MOVL C00760 V=800.0 PL=0
MOVL C00761 V=800.0 PL=0
MOVL C00762 V=800.0 PL=0
MOVL C00763 V=800.0 PL=0
MOVL C00764 V=800.0 PL=0
MOVL C00765 V=800.0 PL=0
MOVL C00766 V=800.0 PL=0
MOVL C00767 V=800.0 PL=0
MOVL C00768 V=800.0 PL=0
MOVL C00769 V=800.0 PL=0
MOVL C00770 V=800.0 PL=0
MOVL C00771 V=800.0 PL=0
MOVL C00772 V=800.0 PL=0
MOVL C00773 V=800.0 PL=0
MOVL C00774 V=800.0 PL=0
MOVL C00775 V=800.0 PL=0
MOVL C00776 V=800.0 PL=0
MOVL C00777 V=800.0 PL=0
MOVL C00778 V=800.0 PL=0
MOVL C00779 V=800.0 PL=0
MOVL C00780 V=800.0 PL=0
MOVL C00781 V=800.0 PL=0
MOVL C00782 V=800.0 PL=0
MOVL C00783 V=800.0 PL=0
MOVL C00784 V=800.0 PL=0
MOVL C00785 V=800.0 PL=0
MOVL C00786 V=800.0 PL=0
MOVL C00787 V=800.0 PL=0
MOVL C00788 V=800.0 PL=0
MOVL C00789 V=800.0 PL=0
MOVL C00790 V=800.0 PL=0
MOVL C00791 V=800.0 PL=0
MOVL C00792 V=800.0 PL=0
MOVL C00793 V=800.0 PL=0
MOVL C00794 V=800.0 PL=0
MOVL C00795 V=800.0 PL=0
MOVL C00796 V=800.0 PL=0
MOVL C00797 V=800.0 PL=0
MOVL C00798 V=800.0 PL=0
MOVL C00799 V=800.0 PL=0
MOVL C00800 V=800.0 PL=0
MOVL C00801 V=800.0 PL=0
MOVL C00802 V=800.0 PL=0
MOVL C00803 V=800.0 PL=0
MOVL C00804 V=800.0 PL=0
MOVL C00805 V=800.0 PL=0
MOVL C00806 V=800.0 PL=0
MOVL C00807 V=800.0 PL=0
MOVL C00808 V=800.0 PL=0
MOVL C00809 V=800.0 PL=0
MOVL C00810 V=800.0 PL=0
MOVL C00811 V=800.0 PL=0
MOVL C00812 V=800.0 PL=0
MOVL C00813 V=800.0 PL=0
MOVL C00814 V=800.0 PL=0
MOVL C00815 V=800.0 PL=0
MOVL C00816 V=800.0 PL=0
MOVL C00817 V=800.0 PL=0
MOVL C00818 V=800.0 PL=0
MOVL C00819 V=800.0 PL=0
MOVL C00820 V=800.0 PL=0
MOVL C00821 V=800.0 PL=0
MOVL C00822 V=800.0 PL=0
MOVL C00823 V=800.0 PL=0
MOVL C00824 V=800.0 PL=0
MOVL C00825 V=800.0 PL=0
MOVL C00826 V=800.0 PL=0
MOVL C00827 V=800.0 PL=0
MOVL C00828 V=800.0 PL=0
MOVL C00829 V=800.0 PL=0
MOVL C00830 V=800.0 PL=0
MOVL C00831 V=800.0 PL=0
MOVL C00832 V=800.0 PL=0
MOVL C00833 V=800.0 PL=0
MOVL C00834 V=800.0 PL=0
MOVL C00835 V=800.0 PL=0
MOVL C00836 V=800.0 PL=0
MOVL C00837 V=800.0 PL=0
MOVL C00838 V=800.0 PL=0
MOVL C00839 V=800.0 PL=0
MOVL C00840 V=800.0 PL=0
MOVL C00841 V=800.0 PL=0
MOVL C00842 V=800.0 PL=0
MOVL C00843 V=800.0 PL=0
MOVL C00844 V=800.0 PL=0
MOVL C00845 V=800.0 PL=0
MOVL C00846 V=800.0 PL=0
MOVL C00847 V=800.0 PL=0
MOVL C00848 V=800.0 PL=0
MOVL C00849 V=800.0 PL=0
MOVL C00850 V=800.0 PL=0
MOVL C00851 V=800.0 PL=0
MOVL C00852 V=800.0 PL=0
MOVL C00853 V=800.0 PL=0
MOVL C00854 V=800.0 PL=0
MOVL C00855 V=800.0 PL=0
MOVL C00856 V=800.0 PL=0
MOVL C00857 V=800.0 PL=0
MOVL C00858 V=800.0 PL=0
MOVL C00859 V=800.0 PL=0
MOVL C00860 V=800.0 PL=0
MOVL C00861 V=800.0 PL=0
MOVL C00862 V=800.0 PL=0
MOVL C00863 V=800.0 PL=0
MOVL C00864 V=800.0 PL=0
MOVL C00865 V=800.0 PL=0
MOVL C00866 V=800.0 PL=0
MOVL C00867 V=800.0 PL=0
MOVL C00868 V=800.0 PL=0
MOVL C00869 V=800.0 PL=0
MOVL C00870 V=800.0 PL=0
MOVL C00871 V=800.0 PL=0
MOVL C00872 V=800.0 PL=0
MOVL C00873 V=800.0 PL=0
MOVL C00874 V=800.0 PL=0
MOVL C00875 V=800.0 PL=0
MOVL C00876 V=800.0 PL=0
MOVL C00877 V=800.0 PL=0
MOVL C00878 V=800.0 PL=0
MOVL C00879 V=800.0 PL=0
MOVL C00880 V=800.0 PL=0
MOVL C00881 V=800.0 PL=0
MOVL C00882 V=800.0 PL=0
MOVL C00883 V=800.0 PL=0
MOVL C00884 V=800.0 PL=0
MOVL C00885 V=800.0 PL=0
MOVL C00886 V=800.0 PL=0
MOVL C00887 V=800.0 PL=0
MOVL C00888 V=800.0 PL=0
MOVL C00889 V=800.0 PL=0
MOVL C00890 V=800.0 PL=0
MOVL C00891 V=800.0 PL=0
MOVL C00892 V=800.0 PL=0
MOVL C00893 V=800.0 PL=0
MOVL C00894 V=800.0 PL=0
MOVL C00895 V=800.0 PL=0
MOVL C00896 V=800.0 PL=0
MOVL C00897 V=800.0 PL=0
MOVL C00898 V=800.0 PL=0
MOVL C00899 V=800.0 PL=0
MOVL C00900 V=800.0 PL=0
MOVL C00901 V=800.0 PL=0
MOVL C00902 V=800.0 PL=0
MOVL C00903 V=800.0 PL=0
MOVL C00904 V=800.0 PL=0
MOVL C00905 V=800.0 PL=0
MOVL C00906 V=800.0 PL=0
MOVL C00907 V=800.0 PL=0
MOVL C00908 V=800.0 PL=0
MOVL C00909 V=800.0 PL=0
MOVL C00910 V=800.0 PL=0
MOVL C00911 V=800.0 PL=0
MOVL C00912 V=800.0 PL=0
MOVL C00913 V=800.0 PL=0
MOVL C00914 V=800.0 PL=0
MOVL C00915 V=800.0 PL=0
MOVL C00916 V=800.0 PL=0
MOVL C00917 V=800.0 PL=0
MOVL C00918 V=800.0 PL=0
MOVL C00919 V=800.0 PL=0
MOVL C00920 V=800.0 PL=0
MOVL C00921 V=800.0 PL=0
MOVL C00922 V=800.0 PL=0
MOVL C00923 V=800.0 PL=0
MOVL C00924 V=800.0 PL=0
MOVL C00925 V=800.0 PL=0
MOVL C00926 V=800.0 PL=0
MOVL C00927 V=800.0 PL=0
MOVL C00928 V=800.0 PL=0
MOVL C00929 V=800.0 PL=0
MOVL C00930 V=800.0 PL=0
MOVL C00931 V=800.0 PL=0
MOVL C00932 V=800.0 PL=0
MOVL C00933 V=800.0 PL=0
MOVL C00934 V=800.0 PL=0
MOVL C00935 V=800.0 PL=0
MOVL C00936 V=800.0 PL=0
MOVL C00937 V=800.0 PL=0
MOVL C00938 V=800.0 PL=0
MOVL C00939 V=800.0 PL=0
MOVL C00940 V=800.0 PL=0
MOVL C00941 V=800.0 PL=0
MOVL C00942 V=800.0 PL=0
MOVL C00943 V=800.0 PL=0
MOVL C00944 V=800.0 PL=0
MOVL C00945 V=800.0 PL=0
MOVL C00946 V=800.0 PL=0
MOVL C00947 V=800.0 PL=0
MOVL C00948 V=800.0 PL=0
MOVL C00949 V=800.0 PL=0
MOVL C00950 V=800.0 PL=0
MOVL C00951 V=800.0 PL=0
MOVL C00952 V=800.0 PL=0
MOVL C00953 V=800.0 PL=0
MOVL C00954 V=800.0 PL=0
MOVL C00955 V=800.0 PL=0
MOVL C00956 V=800.0 PL=0
MOVL C00957 V=800.0 PL=0
MOVL C00958 V=800.0 PL=0
MOVL C00959 V=800.0 PL=0
MOVL C00960 V=800.0 PL=0
MOVL C00961 V=800.0 PL=0
MOVL C00962 V=800.0 PL=0
MOVL C00963 V=800.0 PL=0
MOVL C00964 V=800.0 PL=0
MOVL C00965 V=800.0 PL=0
MOVL C00966 V=800.0 PL=0
MOVL C00967 V=800.0 PL=0
MOVL C00968 V=800.0 PL=0
MOVL C00969 V=800.0 PL=0
MOVL C00970 V=800.0 PL=0
MOVL C00971 V=800.0 PL=0
MOVL C00972 V=800.0 PL=0
MOVL C00973 V=800.0 PL=0
MOVL C00974 V=800.0 PL=0
MOVL C00975 V=800.0 PL=0
MOVL C00976 V=800.0 PL=0
MOVL C00977 V=800.0 PL=0
MOVL C00978 V=800.0 PL=0
MOVL C00979 V=800.0 PL=0
MOVL C00980 V=800.0 PL=0
MOVL C00981 V=800.0 PL=0
MOVL C00982 V=800.0 PL=0
MOVL C00983 V=800.0 PL=0
MOVL C00984 V=800.0 PL=0
MOVL C00985 V=800.0 PL=0
MOVL C00986 V=800.0 PL=0
MOVL C00987 V=800.0 PL=0
MOVL C00988 V=800.0 PL=0
MOVL C00989 V=800.0 PL=0
MOVL C00990 V=800.0 PL=0
MOVL C00991 V=800.0 PL=0
MOVL C00992 V=800.0 PL=0
MOVL C00993 V=800.0 PL=0
MOVL C00994 V=800.0 PL=0
MOVL C00995 V=800.0 PL=0
MOVL C00996 V=800.0 PL=0
MOVL C00997 V=800.0 PL=0
MOVL C00998 V=800.0 PL=0
MOVL C00999 V=800.0 PL=0
MOVL C01000 V=800.0 PL=0
MOVL C01001 V=800.0 PL=0
MOVL C01002 V=800.0 PL=0
MOVL C01003 V=800.0 PL=0
MOVL C01004 V=800.0 PL=0
MOVL C01005 V=800.0 PL=0
MOVL C01006 V=800.0 PL=0
MOVL C01007 V=800.0 PL=0
MOVL C01008 V=800.0 PL=0
MOVL C01009 V=800.0 PL=0
MOVL C01010 V=800.0 PL=0
MOVL C01011 V=800.0 PL=0
MOVL C01012 V=800.0 PL=0
MOVL C01013 V=800.0 PL=0
MOVL C01014 V=800.0 PL=0
MOVL C01015 V=800.0 PL=0
MOVL C01016 V=800.0 PL=0
MOVL C01017 V=800.0 PL=0
MOVL C01018 V=800.0 PL=0
MOVL C01019 V=800.0 PL=0
MOVL C01020 V=800.0 PL=0
MOVL C01021 V=800.0 PL=0
MOVL C01022 V=800.0 PL=0
MOVL C01023 V=800.0 PL=0
MOVL C01024 V=800.0 PL=0
MOVL C01025 V=800.0 PL=0
MOVL C01026 V=800.0 PL=0
MOVL C01027 V=800.0 PL=0
MOVL C01028 V=800.0 PL=0
MOVL C01029 V=800.0 PL=0
MOVL C01030 V=800.0 PL=0
MOVL C01031 V=800.0 PL=0
MOVL C01032 V=800.0 PL=0
MOVL C01033 V=800.0 PL=0
MOVL C01034 V=800.0 PL=0
MOVL C01035 V=800.0 PL=0
MOVL C01036 V=800.0 PL=0
MOVL C01037 V=800.0 PL=0
MOVL C01038 V=800.0 PL=0
MOVL C01039 V=800.0 PL=0
MOVL C01040 V=800.0 PL=0
MOVL C01041 V=800.0 PL=0
MOVL C01042 V=800.0 PL=0
MOVL C01043 V=800.0 PL=0
MOVL C01044 V=800.0 PL=0
MOVL C01045 V=800.0 PL=0
MOVL C01046 V=800.0 PL=0
MOVL C01047 V=800.0 PL=0
MOVL C01048 V=800.0 PL=0
MOVL C01049 V=800.0 PL=0
MOVL C01050 V=800.0 PL=0
MOVL C01051 V=800.0 PL=0
MOVL C01052 V=800.0 PL=0
MOVL C01053 V=800.0 PL=0
MOVL C01054 V=800.0 PL=0
MOVL C01055 V=800.0 PL=0
MOVL C01056 V=800.0 PL=0
MOVL C01057 V=800.0 PL=0
MOVL C01058 V=800.0 PL=0
MOVL C01059 V=800.0 PL=0
MOVL C01060 V=800.0 PL=0
MOVL C01061 V=800.0 PL=0
MOVL C01062 V=800.0 PL=0
MOVL C01063 V=800.0 PL=0
MOVL C01064 V=800.0 PL=0
MOVL C01065 V=800.0 PL=0
MOVL C01066 V=800.0 PL=0
MOVL C01067 V=800.0 PL=0
MOVL C01068 V=800.0 PL=0
MOVL C01069 V=800.0 PL=0
MOVL C01070 V=800.0 PL=0
MOVL C01071 V=800.0 PL=0
MOVL C01072 V=800.0 PL=0
MOVL C01073 V=800.0 PL=0
MOVL C01074 V=800.0 PL=0
MOVL C01075 V=800.0 PL=0
MOVL C01076 V=800.0 PL=0
MOVL C01077 V=800.0 PL=0
MOVL C01078 V=800.0 PL=0
MOVL C01079 V=800.0 PL=0
MOVL C01080 V=800.0 PL=0
MOVL C01081 V=800.0 PL=0
MOVL C01082 V=800.0 PL=0
MOVL C01083 V=800.0 PL=0
MOVL C01084 V=800.0 PL=0
MOVL C01085 V=800.0 PL=0
MOVL C01086 V=800.0 PL=0
MOVL C01087 V=800.0 PL=0
MOVL C01088 V=800.0 PL=0
MOVL C01089 V=800.0 PL=0
MOVL C01090 V=800.0 PL=0
MOVL C01091 V=800.0 PL=0
MOVL C01092 V=800.0 PL=0
MOVL C01093 V=800.0 PL=0
MOVL C01094 V=800.0 PL=0
MOVL C01095 V=800.0 PL=0
MOVL C01096 V=800.0 PL=0
MOVL C01097 V=800.0 PL=0
MOVL C01098 V=800.0 PL=0
MOVL C01099 V=800.0 PL=0
MOVL C01100 V=800.0 PL=0
MOVL C01101 V=800.0 PL=0
MOVL C01102 V=800.0 PL=0
MOVL C01103 V=800.0 PL=0
MOVL C01104 V=800.0 PL=0
MOVL C01105 V=800.0 PL=0
MOVL C01106 V=800.0 PL=0
MOVL C01107 V=800.0 PL=0
MOVL C01108 V=800.0 PL=0
MOVL C01109 V=800.0 PL=0
MOVL C01110 V=800.0 PL=0
MOVL C01111 V=800.0 PL=0
MOVL C01112 V=800.0 PL=0
MOVL C01113 V=800.0 PL=0
MOVL C01114 V=800.0 PL=0
MOVL C01115 V=800.0 PL=0
MOVL C01116 V=800.0 PL=0
MOVL C01117 V=800.0 PL=0
MOVL C01118 V=800.0 PL=0
MOVL C01119 V=800.0 PL=0
MOVL C01120 V=800.0 PL=0
MOVL C01121 V=800.0 PL=0
MOVL C01122 V=800.0 PL=0
MOVL C01123 V=800.0 PL=0
MOVL C01124 V=800.0 PL=0
MOVL C01125 V=800.0 PL=0
MOVL C01126 V=800.0 PL=0
MOVL C01127 V=800.0 PL=0
MOVL C01128 V=800.0 PL=0
MOVL C01129 V=800.0 PL=0
MOVL C01130 V=800.0 PL=0
MOVL C01131 V=800.0 PL=0
MOVL C01132 V=800.0 PL=0
MOVL C01133 V=800.0 PL=0
MOVL C01134 V=800.0 PL=0
MOVL C01135 V=800.0 PL=0
MOVL C01136 V=800.0 PL=0
MOVL C01137 V=800.0 PL=0
MOVL C01138 V=800.0 PL=0
MOVL C01139 V=800.0 PL=0
MOVL C01140 V=800.0 PL=0
MOVL C01141 V=800.0 PL=0
MOVL C01142 V=800.0 PL=0
MOVL C01143 V=800.0 PL=0
MOVL C01144 V=800.0 PL=0
MOVL C01145 V=800.0 PL=0
MOVL C01146 V=800.0 PL=0
MOVL C01147 V=800.0 PL=0
MOVL C01148 V=800.0 PL=0
MOVL C01149 V=800.0 PL=0
MOVL C01150 V=800.0 PL=0
MOVL C01151 V=800.0 PL=0
MOVL C01152 V=800.0 PL=0
MOVL C01153 V=800.0 PL=0
MOVL C01154 V=800.0 PL=0
MOVL C01155 V=800.0 PL=0
MOVL C01156 V=800.0 PL=0
MOVL C01157 V=800.0 PL=0
MOVL C01158 V=800.0 PL=0
MOVL C01159 V=800.0 PL=0
MOVL C01160 V=800.0 PL=0
MOVL C01161 V=800.0 PL=0
MOVL C01162 V=800.0 PL=0
MOVL C01163 V=800.0 PL=0
MOVL C01164 V=800.0 PL=0
MOVL C01165 V=800.0 PL=0
MOVL C01166 V=800.0 PL=0
MOVL C01167 V=800.0 PL=0
MOVL C01168 V=800.0 PL=0
MOVL C01169 V=800.0 PL=0
MOVL C01170 V=800.0 PL=0
MOVL C01171 V=800.0 PL=0
MOVL C01172 V=800.0 PL=0
MOVL C01173 V=800.0 PL=0
MOVL C01174 V=800.0 PL=0
MOVL C01175 V=800.0 PL=0
MOVL C01176 V=800.0 PL=0
MOVL C01177 V=800.0 PL=0
MOVL C01178 V=800.0 PL=0
MOVL C01179 V=800.0 PL=0
MOVL C01180 V=800.0 PL=0
MOVL C01181 V=800.0 PL=0
MOVL C01182 V=800.0 PL=0
MOVL C01183 V=800.0 PL=0
MOVL C01184 V=800.0 PL=0
MOVL C01185 V=800.0 PL=0
MOVL C01186 V=800.0 PL=0
MOVL C01187 V=800.0 PL=0
MOVL C01188 V=800.0 PL=0
MOVL C01189 V=800.0 PL=0
MOVL C01190 V=800.0 PL=0
MOVL C01191 V=800.0 PL=0
MOVL C01192 V=800.0 PL=0
MOVL C01193 V=800.0 PL=0
MOVL C01194 V=800.0 PL=0
MOVL C01195 V=800.0 PL=0
MOVL C01196 V=800.0 PL=0
MOVL C01197 V=800.0 PL=0
MOVL C01198 V=800.0 PL=0
MOVL C01199 V=800.0 PL=0
MOVL C01200 V=800.0 PL=0
MOVL C01201 V=800.0 PL=0
MOVL C01202 V=800.0 PL=0
MOVL C01203 V=800.0 PL=0
MOVL C01204 V=800.0 PL=0
MOVL C01205 V=800.0 PL=0
MOVL C01206 V=800.0 PL=0
MOVL C01207 V=800.0 PL=0
MOVL C01208 V=800.0 PL=0
MOVL C01209 V=800.0 PL=0
MOVL C01210 V=800.0 PL=0
MOVL C01211 V=800.0 PL=0
MOVL C01212 V=800.0 PL=0
MOVL C01213 V=800.0 PL=0
MOVL C01214 V=800.0 PL=0
MOVL C01215 V=800.0 PL=0
MOVL C01216 V=800.0 PL=0
MOVL C01217 V=800.0 PL=0
MOVL C01218 V=800.0 PL=0
MOVL C01219 V=800.0 PL=0
MOVL C01220 V=800.0 PL=0
MOVL C01221 V=800.0 PL=0
MOVL C01222 V=800.0 PL=0
MOVL C01223 V=800.0 PL=0
MOVL C01224 V=800.0 PL=0
MOVL C01225 V=800.0 PL=0
MOVL C01226 V=800.0 PL=0
MOVL C01227 V=800.0 PL=0
MOVL C01228 V=800.0 PL=0
MOVL C01229 V=800.0 PL=0
MOVL C01230 V=800.0 PL=0
MOVL C01231 V=800.0 PL=0
MOVL C01232 V=800.0 PL=0
MOVL C01233 V=800.0 PL=0
MOVL C01234 V=800.0 PL=0
MOVL C01235 V=800.0 PL=0
MOVL C01236 V=800.0 PL=0
MOVL C01237 V=800.0 PL=0
MOVL C01238 V=800.0 PL=0
MOVL C01239 V=800.0 PL=0
MOVL C01240 V=800.0 PL=0
MOVL C01241 V=800.0 PL=0
MOVL C01242 V=800.0 PL=0
MOVL C01243 V=800.0 PL=0
MOVL C01244 V=800.0 PL=0
MOVL C01245 V=800.0 PL=0
MOVL C01246 V=800.0 PL=0
MOVL C01247 V=800.0 PL=0
MOVL C01248 V=800.0 PL=0
MOVL C01249 V=800.0 PL=0
MOVL C01250 V=800.0 PL=0
MOVL C01251 V=800.0 PL=0
MOVL C01252 V=800.0 PL=0
MOVL C01253 V=800.0 PL=0
MOVL C01254 V=800.0 PL=0
MOVL C01255 V=800.0 PL=0
MOVL C01256 V=800.0 PL=0
MOVL C01257 V=800.0 PL=0
MOVL C01258 V=800.0 PL=0
MOVL C01259 V=800.0 PL=0
MOVL C01260 V=800.0 PL=0
MOVL C01261 V=800.0 PL=0
MOVL C01262 V=800.0 PL=0
MOVL C01263 V=800.0 PL=0
MOVL C01264 V=800.0 PL=0
MOVL C01265 V=800.0 PL=0
MOVL C01266 V=800.0 PL=0
MOVL C01267 V=800.0 PL=0
MOVL C01268 V=800.0 PL=0
MOVL C01269 V=800.0 PL=0
MOVL C01270 V=800.0 PL=0
MOVL C01271 V=800.0 PL=0
MOVL C01272 V=800.0 PL=0
MOVL C01273 V=800.0 PL=0
MOVL C01274 V=800.0 PL=0
MOVL C01275 V=800.0 PL=0
MOVL C01276 V=800.0 PL=0
MOVL C01277 V=800.0 PL=0
MOVL C01278 V=800.0 PL=0
MOVL C01279 V=800.0 PL=0
MOVL C01280 V=800.0 PL=0
MOVL C01281 V=800.0 PL=0
MOVL C01282 V=800.0 PL=0
MOVL C01283 V=800.0 PL=0
MOVL C01284 V=800.0 PL=0
MOVL C01285 V=800.0 PL=0
MOVL C01286 V=800.0 PL=0
MOVL C01287 V=800.0 PL=0
MOVL C01288 V=800.0 PL=0
MOVL C01289 V=800.0 PL=0
MOVL C01290 V=800.0 PL=0
MOVL C01291 V=800.0 PL=0
MOVL C01292 V=800.0 PL=0
MOVL C01293 V=800.0 PL=0
MOVL C01294 V=800.0 PL=0
MOVL C01295 V=800.0 PL=0
MOVL C01296 V=800.0 PL=0
MOVL C01297 V=800.0 PL=0
MOVL C01298 V=800.0 PL=0
MOVL C01299 V=800.0 PL=0
MOVL C01300 V=800.0 PL=0
MOVL C01301 V=800.0 PL=0
MOVL C01302 V=800.0 PL=0
MOVL C01303 V=800.0 PL=0
MOVL C01304 V=800.0 PL=0
MOVL C01305 V=800.0 PL=0
MOVL C01306 V=800.0 PL=0
MOVL C01307 V=800.0 PL=0
MOVL C01308 V=800.0 PL=0
MOVL C01309 V=800.0 PL=0
MOVL C01310 V=800.0 PL=0
MOVL C01311 V=800.0 PL=0
MOVL C01312 V=800.0 PL=0
MOVL C01313 V=800.0 PL=0
MOVL C01314 V=800.0 PL=0
MOVL C01315 V=800.0 PL=0
MOVL C01316 V=800.0 PL=0
MOVL C01317 V=800.0 PL=0
MOVL C01318 V=800.0 PL=0
MOVL C01319 V=800.0 PL=0
MOVL C01320 V=800.0 PL=0
MOVL C01321 V=800.0 PL=0
MOVL C01322 V=800.0 PL=0
MOVL C01323 V=800.0 PL=0
MOVL C01324 V=800.0 PL=0
MOVL C01325 V=800.0 PL=0
MOVL C01326 V=800.0 PL=0
MOVL C01327 V=800.0 PL=0
MOVL C01328 V=800.0 PL=0
MOVL C01329 V=800.0 PL=0
MOVL C01330 V=800.0 PL=0
MOVL C01331 V=800.0 PL=0
MOVL C01332 V=800.0 PL=0
MOVL C01333 V=800.0 PL=0
MOVL C01334 V=800.0 PL=0
MOVL C01335 V=800.0 PL=0
MOVL C01336 V=800.0 PL=0
MOVL C01337 V=800.0 PL=0
MOVL C01338 V=800.0 PL=0
MOVL C01339 V=800.0 PL=0
MOVL C01340 V=800.0 PL=0
MOVL C01341 V=800.0 PL=0
MOVL C01342 V=800.0 PL=0
MOVL C01343 V=800.0 PL=0
MOVL C01344 V=800.0 PL=0
MOVL C01345 V=800.0 PL=0
MOVL C01346 V=800.0 PL=0
MOVL C01347 V=800.0 PL=0
MOVL C01348 V=800.0 PL=0
MOVL C01349 V=800.0 PL=0
MOVL C01350 V=800.0 PL=0
MOVL C01351 V=800.0 PL=0
MOVL C01352 V=800.0 PL=0
MOVL C01353 V=800.0 PL=0
MOVL C01354 V=800.0 PL=0
MOVL C01355 V=800.0 PL=0
MOVL C01356 V=800.0 PL=0
MOVL C01357 V=800.0 PL=0
MOVL C01358 V=800.0 PL=0
MOVL C01359 V=800.0 PL=0
MOVL C01360 V=800.0 PL=0
MOVL C01361 V=800.0 PL=0
MOVL C01362 V=800.0 PL=0
MOVL C01363 V=800.0 PL=0
MOVL C01364 V=800.0 PL=0
MOVL C01365 V=800.0 PL=0
MOVL C01366 V=800.0 PL=0
MOVL C01367 V=800.0 PL=0
MOVL C01368 V=800.0 PL=0
MOVL C01369 V=800.0 PL=0
MOVL C01370 V=800.0 PL=0
MOVL C01371 V=800.0 PL=0
MOVL C01372 V=800.0 PL=0
MOVL C01373 V=800.0 PL=0
MOVL C01374 V=800.0 PL=0
MOVL C01375 V=800.0 PL=0
MOVL C01376 V=800.0 PL=0
MOVL C01377 V=800.0 PL=0
MOVL C01378 V=800.0 PL=0
MOVL C01379 V=800.0 PL=0
MOVL C01380 V=800.0 PL=0
MOVL C01381 V=800.0 PL=0
MOVL C01382 V=800.0 PL=0
MOVL C01383 V=800.0 PL=0
MOVL C01384 V=800.0 PL=0
MOVL C01385 V=800.0 PL=0
MOVL C01386 V=800.0 PL=0
MOVL C01387 V=800.0 PL=0
MOVL C01388 V=800.0 PL=0
MOVL C01389 V=800.0 PL=0
MOVL C01390 V=800.0 PL=0
MOVL C01391 V=800.0 PL=0
MOVL C01392 V=800.0 PL=0
MOVL C01393 V=800.0 PL=0
MOVL C01394 V=800.0 PL=0
MOVL C01395 V=800.0 PL=0
MOVL C01396 V=800.0 PL=0
MOVL C01397 V=800.0 PL=0
MOVL C01398 V=800.0 PL=0
MOVL C01399 V=800.0 PL=0
MOVL C01400 V=800.0 PL=0
MOVL C01401 V=800.0 PL=0
MOVL C01402 V=800.0 PL=0
MOVL C01403 V=800.0 PL=0
MOVL C01404 V=800.0 PL=0
MOVL C01405 V=800.0 PL=0
MOVL C01406 V=800.0 PL=0
MOVL C01407 V=800.0 PL=0
MOVL C01408 V=800.0 PL=0
MOVL C01409 V=800.0 PL=0
MOVL C01410 V=800.0 PL=0
MOVL C01411 V=800.0 PL=0
MOVL C01412 V=800.0 PL=0
MOVL C01413 V=800.0 PL=0
MOVL C01414 V=800.0 PL=0
MOVL C01415 V=800.0 PL=0
MOVL C01416 V=800.0 PL=0
MOVL C01417 V=800.0 PL=0
MOVL C01418 V=800.0 PL=0
MOVL C01419 V=800.0 PL=0
MOVL C01420 V=800.0 PL=0
MOVL C01421 V=800.0 PL=0
MOVL C01422 V=800.0 PL=0
MOVL C01423 V=800.0 PL=0
MOVL C01424 V=800.0 PL=0
MOVL C01425 V=800.0 PL=0
MOVL C01426 V=800.0 PL=0
MOVL C01427 V=800.0 PL=0
MOVL C01428 V=800.0 PL=0
MOVL C01429 V=800.0 PL=0
MOVL C01430 V=800.0 PL=0
MOVL C01431 V=800.0 PL=0
MOVL C01432 V=800.0 PL=0
MOVL C01433 V=800.0 PL=0
MOVL C01434 V=800.0 PL=0
MOVL C01435 V=800.0 PL=0
MOVL C01436 V=800.0 PL=0
MOVL C01437 V=800.0 PL=0
MOVL C01438 V=800.0 PL=0
MOVL C01439 V=800.0 PL=0
MOVL C01440 V=800.0 PL=0
MOVL C01441 V=800.0 PL=0
MOVL C01442 V=800.0 PL=0
MOVL C01443 V=800.0 PL=0
MOVL C01444 V=800.0 PL=0
MOVL C01445 V=800.0 PL=0
MOVL C01446 V=800.0 PL=0
MOVL C01447 V=800.0 PL=0
MOVL C01448 V=800.0 PL=0
MOVL C01449 V=800.0 PL=0
MOVL C01450 V=800.0 PL=0
MOVL C01451 V=800.0 PL=0
MOVL C01452 V=800.0 PL=0
MOVL C01453 V=800.0 PL=0
MOVL C01454 V=800.0 PL=0
MOVL C01455 V=800.0 PL=0
MOVL C01456 V=800.0 PL=0
MOVL C01457 V=800.0 PL=0
MOVL C01458 V=800.0 PL=0
MOVL C01459 V=800.0 PL=0
MOVL C01460 V=800.0 PL=0
MOVL C01461 V=800.0 PL=0
MOVL C01462 V=800.0 PL=0
MOVL C01463 V=800.0 PL=0
MOVL C01464 V=800.0 PL=0
MOVL C01465 V=800.0 PL=0
MOVL C01466 V=800.0 PL=0
MOVL C01467 V=800.0 PL=0
MOVL C01468 V=800.0 PL=0
MOVL C01469 V=800.0 PL=0
MOVL C01470 V=800.0 PL=0
MOVL C01471 V=800.0 PL=0
MOVL C01472 V=800.0 PL=0
MOVL C01473 V=800.0 PL=0
MOVL C01474 V=800.0 PL=0
MOVL C01475 V=800.0 PL=0
MOVL C01476 V=800.0 PL=0
MOVL C01477 V=800.0 PL=0
MOVL C01478 V=800.0 PL=0
MOVL C01479 V=800.0 PL=0
MOVL C01480 V=800.0 PL=0
MOVL C01481 V=800.0 PL=0
MOVL C01482 V=800.0 PL=0
MOVL C01483 V=800.0 PL=0
MOVL C01484 V=800.0 PL=0
MOVL C01485 V=800.0 PL=0
MOVL C01486 V=800.0 PL=0
MOVL C01487 V=800.0 PL=0
MOVL C01488 V=800.0 PL=0
MOVL C01489 V=800.0 PL=0
MOVL C01490 V=800.0 PL=0
MOVL C01491 V=800.0 PL=0
MOVL C01492 V=800.0 PL=0
MOVL C01493 V=800.0 PL=0
MOVL C01494 V=800.0 PL=0
MOVL C01495 V=800.0 PL=0
MOVL C01496 V=800.0 PL=0
MOVL C01497 V=800.0 PL=0
MOVL C01498 V=800.0 PL=0
MOVL C01499 V=800.0 PL=0
MOVL C01500 V=800.0 PL=0
MOVL C01501 V=800.0 PL=0
MOVL C01502 V=800.0 PL=0
MOVL C01503 V=800.0 PL=0
MOVL C01504 V=800.0 PL=0
MOVL C01505 V=800.0 PL=0
MOVL C01506 V=800.0 PL=0
MOVL C01507 V=800.0 PL=0
MOVL C01508 V=800.0 PL=0
MOVL C01509 V=800.0 PL=0
MOVL C01510 V=800.0 PL=0
MOVL C01511 V=800.0 PL=0
MOVL C01512 V=800.0 PL=0
MOVL C01513 V=800.0 PL=0
MOVL C01514 V=800.0 PL=0
MOVL C01515 V=800.0 PL=0
MOVL C01516 V=800.0 PL=0
MOVL C01517 V=800.0 PL=0
MOVL C01518 V=800.0 PL=0
MOVL C01519 V=800.0 PL=0
MOVL C01520 V=800.0 PL=0
MOVL C01521 V=800.0 PL=0
MOVL C01522 V=800.0 PL=0
MOVL C01523 V=800.0 PL=0
MOVL C01524 V=800.0 PL=0
MOVL C01525 V=800.0 PL=0
MOVL C01526 V=800.0 PL=0
MOVL C01527 V=800.0 PL=0
MOVL C01528 V=800.0 PL=0
MOVL C01529 V=800.0 PL=0
MOVL C01530 V=800.0 PL=0
MOVL C01531 V=800.0 PL=0
MOVL C01532 V=800.0 PL=0
MOVL C01533 V=800.0 PL=0
MOVL C01534 V=800.0 PL=0
MOVL C01535 V=800.0 PL=0
MOVL C01536 V=800.0 PL=0
MOVL C01537 V=800.0 PL=0
MOVL C01538 V=800.0 PL=0
MOVL C01539 V=800.0 PL=0
MOVL C01540 V=800.0 PL=0
MOVL C01541 V=800.0 PL=0
MOVL C01542 V=800.0 PL=0
MOVL C01543 V=800.0 PL=0
MOVL C01544 V=800.0 PL=0
MOVL C01545 V=800.0 PL=0
MOVL C01546 V=800.0 PL=0
MOVL C01547 V=800.0 PL=0
MOVL C01548 V=800.0 PL=0
MOVL C01549 V=800.0 PL=0
MOVL C01550 V=800.0 PL=0
MOVL C01551 V=800.0 PL=0
MOVL C01552 V=800.0 PL=0
MOVL C01553 V=800.0 PL=0
MOVL C01554 V=800.0 PL=0
MOVL C01555 V=800.0 PL=0
MOVL C01556 V=800.0 PL=0
MOVL C01557 V=800.0 PL=0
MOVL C01558 V=800.0 PL=0
MOVL C01559 V=800.0 PL=0
MOVL C01560 V=800.0 PL=0
MOVL C01561 V=800.0 PL=0
MOVL C01562 V=800.0 PL=0
MOVL C01563 V=800.0 PL=0
MOVL C01564 V=800.0 PL=0
MOVL C01565 V=800.0 PL=0
MOVL C01566 V=800.0 PL=0
MOVL C01567 V=800.0 PL=0
MOVL C01568 V=800.0 PL=0
MOVL C01569 V=800.0 PL=0
MOVL C01570 V=800.0 PL=0
MOVL C01571 V=800.0 PL=0
MOVL C01572 V=800.0 PL=0
MOVL C01573 V=800.0 PL=0
MOVL C01574 V=800.0 PL=0
MOVL C01575 V=800.0 PL=0
MOVL C01576 V=800.0 PL=0
MOVL C01577 V=800.0 PL=0
MOVL C01578 V=800.0 PL=0
MOVL C01579 V=800.0 PL=0
MOVL C01580 V=800.0 PL=0
MOVL C01581 V=800.0 PL=0
MOVL C01582 V=800.0 PL=0
MOVL C01583 V=800.0 PL=0
MOVL C01584 V=800.0 PL=0
MOVL C01585 V=800.0 PL=0
MOVL C01586 V=800.0 PL=0
MOVL C01587 V=800.0 PL=0
MOVL C01588 V=800.0 PL=0
MOVL C01589 V=800.0 PL=0
MOVL C01590 V=800.0 PL=0
MOVL C01591 V=800.0 PL=0
MOVL C01592 V=800.0 PL=0
MOVL C01593 V=800.0 PL=0
MOVL C01594 V=800.0 PL=0
MOVL C01595 V=800.0 PL=0
MOVL C01596 V=800.0 PL=0
MOVL C01597 V=800.0 PL=0
MOVL C01598 V=800.0 PL=0
MOVL C01599 V=800.0 PL=0
MOVL C01600 V=800.0 PL=0
MOVL C01601 V=800.0 PL=0
MOVL C01602 V=800.0 PL=0
MOVL C01603 V=800.0 PL=0
MOVL C01604 V=800.0 PL=0
MOVL C01605 V=800.0 PL=0
MOVL C01606 V=800.0 PL=0
MOVL C01607 V=800.0 PL=0
MOVL C01608 V=800.0 PL=0
MOVL C01609 V=800.0 PL=0
MOVL C01610 V=800.0 PL=0
MOVL C01611 V=800.0 PL=0
MOVL C01612 V=800.0 PL=0
MOVL C01613 V=800.0 PL=0
MOVL C01614 V=800.0 PL=0
MOVL C01615 V=800.0 PL=0
MOVL C01616 V=800.0 PL=0
MOVL C01617 V=800.0 PL=0
MOVL C01618 V=800.0 PL=0
MOVL C01619 V=800.0 PL=0
MOVL C01620 V=800.0 PL=0
MOVL C01621 V=800.0 PL=0
MOVL C01622 V=800.0 PL=0
MOVL C01623 V=800.0 PL=0
MOVL C01624 V=800.0 PL=0
MOVL C01625 V=800.0 PL=0
MOVL C01626 V=800.0 PL=0
MOVL C01627 V=800.0 PL=0
MOVL C01628 V=800.0 PL=0
MOVL C01629 V=800.0 PL=0
MOVL C01630 V=800.0 PL=0
MOVL C01631 V=800.0 PL=0
MOVL C01632 V=800.0 PL=0
MOVL C01633 V=800.0 PL=0
MOVL C01634 V=800.0 PL=0
MOVL C01635 V=800.0 PL=0
MOVL C01636 V=800.0 PL=0
MOVL C01637 V=800.0 PL=0
MOVL C01638 V=800.0 PL=0
MOVL C01639 V=800.0 PL=0
MOVL C01640 V=800.0 PL=0
MOVL C01641 V=800.0 PL=0
MOVL C01642 V=800.0 PL=0
MOVL C01643 V=800.0 PL=0
MOVL C01644 V=800.0 PL=0
MOVL C01645 V=800.0 PL=0
MOVL C01646 V=800.0 PL=0
MOVL C01647 V=800.0 PL=0
MOVL C01648 V=800.0 PL=0
MOVL C01649 V=800.0 PL=0
MOVL C01650 V=800.0 PL=0
MOVL C01651 V=800.0 PL=0
MOVL C01652 V=800.0 PL=0
MOVL C01653 V=800.0 PL=0
MOVL C01654 V=800.0 PL=0
MOVL C01655 V=800.0 PL=0
MOVL C01656 V=800.0 PL=0
MOVL C01657 V=800.0 PL=0
MOVL C01658 V=800.0 PL=0
MOVL C01659 V=800.0 PL=0
MOVL C01660 V=800.0 PL=0
MOVL C01661 V=800.0 PL=0
MOVL C01662 V=800.0 PL=0
MOVL C01663 V=800.0 PL=0
MOVL C01664 V=800.0 PL=0
MOVL C01665 V=800.0 PL=0
MOVL C01666 V=800.0 PL=0
MOVL C01667 V=800.0 PL=0
MOVL C01668 V=800.0 PL=0
MOVL C01669 V=800.0 PL=0
MOVL C01670 V=800.0 PL=0
MOVL C01671 V=800.0 PL=0
MOVL C01672 V=800.0 PL=0
MOVL C01673 V=800.0 PL=0
MOVL C01674 V=800.0 PL=0
MOVL C01675 V=800.0 PL=0
MOVL C01676 V=800.0 PL=0
MOVL C01677 V=800.0 PL=0
MOVL C01678 V=800.0 PL=0
MOVL C01679 V=800.0 PL=0
MOVL C01680 V=800.0 PL=0
MOVL C01681 V=800.0 PL=0
MOVL C01682 V=800.0 PL=0
MOVL C01683 V=800.0 PL=0
MOVL C01684 V=800.0 PL=0
MOVL C01685 V=800.0 PL=0
MOVL C01686 V=800.0 PL=0
MOVL C01687 V=800.0 PL=0
MOVL C01688 V=800.0 PL=0
MOVL C01689 V=800.0 PL=0
MOVL C01690 V=800.0 PL=0
MOVL C01691 V=800.0 PL=0
MOVL C01692 V=800.0 PL=0
MOVL C01693 V=800.0 PL=0
MOVL C01694 V=800.0 PL=0
MOVL C01695 V=800.0 PL=0
MOVL C01696 V=800.0 PL=0
MOVL C01697 V=800.0 PL=0
MOVL C01698 V=800.0 PL=0
MOVL C01699 V=800.0 PL=0
MOVL C01700 V=800.0 PL=0
MOVL C01701 V=800.0 PL=0
MOVL C01702 V=800.0 PL=0
MOVL C01703 V=800.0 PL=0
MOVL C01704 V=800.0 PL=0
MOVL C01705 V=800.0 PL=0
MOVL C01706 V=800.0 PL=0
MOVL C01707 V=800.0 PL=0
MOVL C01708 V=800.0 PL=0
MOVL C01709 V=800.0 PL=0
MOVL C01710 V=800.0 PL=0
MOVL C01711 V=800.0 PL=0
MOVL C01712 V=800.0 PL=0
MOVL C01713 V=800.0 PL=0
MOVL C01714 V=800.0 PL=0
MOVL C01715 V=800.0 PL=0
MOVL C01716 V=800.0 PL=0
MOVL C01717 V=800.0 PL=0
MOVL C01718 V=800.0 PL=0
MOVL C01719 V=800.0 PL=0
MOVL C01720 V=800.0 PL=0
MOVL C01721 V=800.0 PL=0
MOVL C01722 V=800.0 PL=0
MOVL C01723 V=800.0 PL=0
MOVL C01724 V=800.0 PL=0
MOVL C01725 V=800.0 PL=0
MOVL C01726 V=800.0 PL=0
MOVL C01727 V=800.0 PL=0
MOVL C01728 V=800.0 PL=0
MOVL C01729 V=800.0 PL=0
MOVL C01730 V=800.0 PL=0
MOVL C01731 V=800.0 PL=0
MOVL C01732 V=800.0 PL=0
MOVL C01733 V=800.0 PL=0
MOVL C01734 V=800.0 PL=0
MOVL C01735 V=800.0 PL=0
MOVL C01736 V=800.0 PL=0
MOVL C01737 V=800.0 PL=0
MOVL C01738 V=800.0 PL=0
MOVL C01739 V=800.0 PL=0
MOVL C01740 V=800.0 PL=0
MOVL C01741 V=800.0 PL=0
MOVL C01742 V=800.0 PL=0
MOVL C01743 V=800.0 PL=0
MOVL C01744 V=800.0 PL=0
MOVL C01745 V=800.0 PL=0
MOVL C01746 V=800.0 PL=0
MOVL C01747 V=800.0 PL=0
MOVL C01748 V=800.0 PL=0
MOVL C01749 V=800.0 PL=0
MOVL C01750 V=800.0 PL=0
MOVL C01751 V=800.0 PL=0
MOVL C01752 V=800.0 PL=0
MOVL C01753 V=800.0 PL=0
MOVL C01754 V=800.0 PL=0
MOVL C01755 V=800.0 PL=0
MOVL C01756 V=800.0 PL=0
MOVL C01757 V=800.0 PL=0
MOVL C01758 V=800.0 PL=0
MOVL C01759 V=800.0 PL=0
MOVL C01760 V=800.0 PL=0
MOVL C01761 V=800.0 PL=0
MOVL C01762 V=800.0 PL=0
MOVL C01763 V=800.0 PL=0
MOVL C01764 V=800.0 PL=0
MOVL C01765 V=800.0 PL=0
MOVL C01766 V=800.0 PL=0
MOVL C01767 V=800.0 PL=0
MOVL C01768 V=800.0 PL=0
MOVL C01769 V=800.0 PL=0
MOVL C01770 V=800.0 PL=0
MOVL C01771 V=800.0 PL=0
MOVL C01772 V=800.0 PL=0
MOVL C01773 V=800.0 PL=0
MOVL C01774 V=800.0 PL=0
MOVL C01775 V=800.0 PL=0
MOVL C01776 V=800.0 PL=0
MOVL C01777 V=800.0 PL=0
MOVL C01778 V=800.0 PL=0
MOVL C01779 V=800.0 PL=0
MOVL C01780 V=800.0 PL=0
MOVL C01781 V=800.0 PL=0
MOVL C01782 V=800.0 PL=0
MOVL C01783 V=800.0 PL=0
MOVL C01784 V=800.0 PL=0
MOVL C01785 V=800.0 PL=0
MOVL C01786 V=800.0 PL=0
MOVL C01787 V=800.0 PL=0
MOVL C01788 V=800.0 PL=0
MOVL C01789 V=800.0 PL=0
MOVL C01790 V=800.0 PL=0
MOVL C01791 V=800.0 PL=0
MOVL C01792 V=800.0 PL=0
MOVL C01793 V=800.0 PL=0
MOVL C01794 V=800.0 PL=0
MOVL C01795 V=800.0 PL=0
MOVL C01796 V=800.0 PL=0
MOVL C01797 V=800.0 PL=0
MOVL C01798 V=800.0 PL=0
MOVL C01799 V=800.0 PL=0
MOVL C01800 V=800.0 PL=0
MOVL C01801 V=800.0 PL=0
MOVL C01802 V=800.0 PL=0
MOVL C01803 V=800.0 PL=0
MOVL C01804 V=800.0 PL=0
MOVL C01805 V=800.0 PL=0
MOVL C01806 V=800.0 PL=0
MOVL C01807 V=800.0 PL=0
MOVL C01808 V=800.0 PL=0
MOVL C01809 V=800.0 PL=0
MOVL C01810 V=800.0 PL=0
MOVL C01811 V=800.0 PL=0
MOVL C01812 V=800.0 PL=0
MOVL C01813 V=800.0 PL=0
MOVL C01814 V=800.0 PL=0
MOVL C01815 V=800.0 PL=0
MOVL C01816 V=800.0 PL=0
MOVL C01817 V=800.0 PL=0
MOVL C01818 V=800.0 PL=0
MOVL C01819 V=800.0 PL=0
MOVL C01820 V=800.0 PL=0
MOVL C01821 V=800.0 PL=0
MOVL C01822 V=800.0 PL=0
MOVL C01823 V=800.0 PL=0
MOVL C01824 V=800.0 PL=0
MOVL C01825 V=800.0 PL=0
MOVL C01826 V=800.0 PL=0
MOVL C01827 V=800.0 PL=0
MOVL C01828 V=800.0 PL=0
MOVL C01829 V=800.0 PL=0
MOVL C01830 V=800.0 PL=0
MOVL C01831 V=800.0 PL=0
MOVL C01832 V=800.0 PL=0
MOVL C01833 V=800.0 PL=0
MOVL C01834 V=800.0 PL=0
MOVL C01835 V=800.0 PL=0
MOVL C01836 V=800.0 PL=0
MOVL C01837 V=800.0 PL=0
MOVL C01838 V=800.0 PL=0
MOVL C01839 V=800.0 PL=0
MOVL C01840 V=800.0 PL=0
MOVL C01841 V=800.0 PL=0
MOVL C01842 V=800.0 PL=0
MOVL C01843 V=800.0 PL=0
MOVL C01844 V=800.0 PL=0
MOVL C01845 V=800.0 PL=0
MOVL C01846 V=800.0 PL=0
MOVL C01847 V=800.0 PL=0
MOVL C01848 V=800.0 PL=0
MOVL C01849 V=800.0 PL=0
MOVL C01850 V=800.0 PL=0
MOVL C01851 V=800.0 PL=0
MOVL C01852 V=800.0 PL=0
MOVL C01853 V=800.0 PL=0
MOVL C01854 V=800.0 PL=0
MOVL C01855 V=800.0 PL=0
MOVL C01856 V=800.0 PL=0
MOVL C01857 V=800.0 PL=0
MOVL C01858 V=800.0 PL=0
MOVL C01859 V=800.0 PL=0
MOVL C01860 V=800.0 PL=0
MOVL C01861 V=800.0 PL=0
MOVL C01862 V=800.0 PL=0
MOVL C01863 V=800.0 PL=0
MOVL C01864 V=800.0 PL=0
MOVL C01865 V=800.0 PL=0
MOVL C01866 V=800.0 PL=0
MOVL C01867 V=800.0 PL=0
MOVL C01868 V=800.0 PL=0
MOVL C01869 V=800.0 PL=0
MOVL C01870 V=800.0 PL=0
MOVL C01871 V=800.0 PL=0
MOVL C01872 V=800.0 PL=0
MOVL C01873 V=800.0 PL=0
MOVL C01874 V=800.0 PL=0
MOVL C01875 V=800.0 PL=0
MOVL C01876 V=800.0 PL=0
MOVL C01877 V=800.0 PL=0
MOVL C01878 V=800.0 PL=0
MOVL C01879 V=800.0 PL=0
MOVL C01880 V=800.0 PL=0
MOVL C01881 V=800.0 PL=0
MOVL C01882 V=800.0 PL=0
MOVL C01883 V=800.0 PL=0
MOVL C01884 V=800.0 PL=0
MOVL C01885 V=800.0 PL=0
MOVL C01886 V=800.0 PL=0
MOVL C01887 V=800.0 PL=0
MOVL C01888 V=800.0 PL=0
MOVL C01889 V=800.0 PL=0
MOVL C01890 V=800.0 PL=0
MOVL C01891 V=800.0 PL=0
MOVL C01892 V=800.0 PL=0
MOVL C01893 V=800.0 PL=0
MOVL C01894 V=800.0 PL=0
MOVL C01895 V=800.0 PL=0
MOVL C01896 V=800.0 PL=0
MOVL C01897 V=800.0 PL=0
MOVL C01898 V=800.0 PL=0
MOVL C01899 V=800.0 PL=0
MOVL C01900 V=800.0 PL=0
MOVL C01901 V=800.0 PL=0
MOVL C01902 V=800.0 PL=0
MOVL C01903 V=800.0 PL=0
MOVL C01904 V=800.0 PL=0
MOVL C01905 V=800.0 PL=0
MOVL C01906 V=800.0 PL=0
MOVL C01907 V=800.0 PL=0
MOVL C01908 V=800.0 PL=0
MOVL C01909 V=800.0 PL=0
MOVL C01910 V=800.0 PL=0
MOVL C01911 V=800.0 PL=0
MOVL C01912 V=800.0 PL=0
MOVL C01913 V=800.0 PL=0
MOVL C01914 V=800.0 PL=0
MOVL C01915 V=800.0 PL=0
MOVL C01916 V=800.0 PL=0
MOVL C01917 V=800.0 PL=0
MOVL C01918 V=800.0 PL=0
MOVL C01919 V=800.0 PL=0
MOVL C01920 V=800.0 PL=0
MOVL C01921 V=800.0 PL=0
MOVL C01922 V=800.0 PL=0
MOVL C01923 V=800.0 PL=0
MOVL C01924 V=800.0 PL=0
MOVL C01925 V=800.0 PL=0
MOVL C01926 V=800.0 PL=0
MOVL C01927 V=800.0 PL=0
MOVL C01928 V=800.0 PL=0
MOVL C01929 V=800.0 PL=0
MOVL C01930 V=800.0 PL=0
MOVL C01931 V=800.0 PL=0
MOVL C01932 V=800.0 PL=0
MOVL C01933 V=800.0 PL=0
MOVL C01934 V=800.0 PL=0
MOVL C01935 V=800.0 PL=0
MOVL C01936 V=800.0 PL=0
MOVL C01937 V=800.0 PL=0
MOVL C01938 V=800.0 PL=0
MOVL C01939 V=800.0 PL=0
MOVL C01940 V=800.0 PL=0
MOVL C01941 V=800.0 PL=0
MOVL C01942 V=800.0 PL=0
MOVL C01943 V=800.0 PL=0
MOVL C01944 V=800.0 PL=0
MOVL C01945 V=800.0 PL=0
MOVL C01946 V=800.0 PL=0
MOVL C01947 V=800.0 PL=0
MOVL C01948 V=800.0 PL=0
MOVL C01949 V=800.0 PL=0
MOVL C01950 V=800.0 PL=0
MOVL C01951 V=800.0 PL=0
MOVL C01952 V=800.0 PL=0
MOVL C01953 V=800.0 PL=0
MOVL C01954 V=800.0 PL=0
MOVL C01955 V=800.0 PL=0
MOVL C01956 V=800.0 PL=0
MOVL C01957 V=800.0 PL=0
MOVL C01958 V=800.0 PL=0
MOVL C01959 V=800.0 PL=0
MOVL C01960 V=800.0 PL=0
MOVL C01961 V=800.0 PL=0
MOVL C01962 V=800.0 PL=0
MOVL C01963 V=800.0 PL=0
MOVL C01964 V=800.0 PL=0
MOVL C01965 V=800.0 PL=0
MOVL C01966 V=800.0 PL=0
MOVL C01967 V=800.0 PL=0
MOVL C01968 V=800.0 PL=0
MOVL C01969 V=800.0 PL=0
MOVL C01970 V=800.0 PL=0
MOVL C01971 V=800.0 PL=0
MOVL C01972 V=800.0 PL=0
MOVL C01973 V=800.0 PL=0
MOVL C01974 V=800.0 PL=0
MOVL C01975 V=800.0 PL=0
MOVL C01976 V=800.0 PL=0
MOVL C01977 V=800.0 PL=0
MOVL C01978 V=800.0 PL=0
MOVL C01979 V=800.0 PL=0
MOVL C01980 V=800.0 PL=0
MOVL C01981 V=800.0 PL=0
MOVL C01982 V=800.0 PL=0
MOVL C01983 V=800.0 PL=0
MOVL C01984 V=800.0 PL=0
MOVL C01985 V=800.0 PL=0
MOVL C01986 V=800.0 PL=0
MOVL C01987 V=800.0 PL=0
MOVL C01988 V=800.0 PL=0
MOVL C01989 V=800.0 PL=0
MOVL C01990 V=800.0 PL=0
MOVL C01991 V=800.0 PL=0
MOVL C01992 V=800.0 PL=0
MOVL C01993 V=800.0 PL=0
MOVL C01994 V=800.0 PL=0
MOVL C01995 V=800.0 PL=0
MOVL C01996 V=800.0 PL=0
MOVL C01997 V=800.0 PL=0
MOVL C01998 V=800.0 PL=0
MOVL C01999 V=800.0 PL=0
MOVL C02000 V=800.0 PL=0
MOVL C02001 V=800.0 PL=0
MOVL C02002 V=800.0 PL=0
MOVL C02003 V=800.0 PL=0
MOVL C02004 V=800.0 PL=0
MOVL C02005 V=800.0 PL=0
MOVL C02006 V=800.0 PL=0
MOVL C02007 V=800.0 PL=0
MOVL C02008 V=800.0 PL=0
MOVL C02009 V=800.0 PL=0
MOVL C02010 V=800.0 PL=0
MOVL C02011 V=800.0 PL=0
MOVL C02012 V=800.0 PL=0
MOVL C02013 V=800.0 PL=0
MOVL C02014 V=800.0 PL=0
MOVL C02015 V=800.0 PL=0
MOVL C02016 V=800.0 PL=0
MOVL C02017 V=800.0 PL=0
MOVL C02018 V=800.0 PL=0
MOVL C02019 V=800.0 PL=0
MOVL C02020 V=800.0 PL=0
MOVL C02021 V=800.0 PL=0
MOVL C02022 V=800.0 PL=0
MOVL C02023 V=800.0 PL=0
MOVL C02024 V=800.0 PL=0
MOVL C02025 V=800.0 PL=0
MOVL C02026 V=800.0 PL=0
MOVL C02027 V=800.0 PL=0
MOVL C02028 V=800.0 PL=0
MOVL C02029 V=800.0 PL=0
MOVL C02030 V=800.0 PL=0
MOVL C02031 V=800.0 PL=0
MOVL C02032 V=800.0 PL=0
MOVL C02033 V=800.0 PL=0
MOVL C02034 V=800.0 PL=0
MOVL C02035 V=800.0 PL=0
MOVL C02036 V=800.0 PL=0
MOVL C02037 V=800.0 PL=0
MOVL C02038 V=800.0 PL=0
MOVL C02039 V=800.0 PL=0
MOVL C02040 V=800.0 PL=0
MOVL C02041 V=800.0 PL=0
MOVL C02042 V=800.0 PL=0
MOVL C02043 V=800.0 PL=0
MOVL C02044 V=800.0 PL=0
MOVL C02045 V=800.0 PL=0
MOVL C02046 V=800.0 PL=0
MOVL C02047 V=800.0 PL=0
MOVL C02048 V=800.0 PL=0
MOVL C02049 V=800.0 PL=0
MOVL C02050 V=800.0 PL=0
MOVL C02051 V=800.0 PL=0
MOVL C02052 V=800.0 PL=0
MOVL C02053 V=800.0 PL=0
MOVL C02054 V=800.0 PL=0
MOVL C02055 V=800.0 PL=0
MOVL C02056 V=800.0 PL=0
MOVL C02057 V=800.0 PL=0
MOVL C02058 V=800.0 PL=0
MOVL C02059 V=800.0 PL=0
MOVL C02060 V=800.0 PL=0
MOVL C02061 V=800.0 PL=0
MOVL C02062 V=800.0 PL=0
MOVL C02063 V=800.0 PL=0
MOVL C02064 V=800.0 PL=0
MOVL C02065 V=800.0 PL=0
MOVL C02066 V=800.0 PL=0
MOVL C02067 V=800.0 PL=0
MOVL C02068 V=800.0 PL=0
MOVL C02069 V=800.0 PL=0
MOVL C02070 V=800.0 PL=0
MOVL C02071 V=800.0 PL=0
MOVL C02072 V=800.0 PL=0
MOVL C02073 V=800.0 PL=0
MOVL C02074 V=800.0 PL=0
MOVL C02075 V=800.0 PL=0
MOVL C02076 V=800.0 PL=0
MOVL C02077 V=800.0 PL=0
MOVL C02078 V=800.0 PL=0
MOVL C02079 V=800.0 PL=0
MOVL C02080 V=800.0 PL=0
MOVL C02081 V=800.0 PL=0
MOVL C02082 V=800.0 PL=0
MOVL C02083 V=800.0 PL=0
MOVL C02084 V=800.0 PL=0
MOVL C02085 V=800.0 PL=0
MOVL C02086 V=800.0 PL=0
MOVL C02087 V=800.0 PL=0
MOVL C02088 V=800.0 PL=0
MOVL C02089 V=800.0 PL=0
MOVL C02090 V=800.0 PL=0
MOVL C02091 V=800.0 PL=0
MOVL C02092 V=800.0 PL=0
